// TIA Portal V15.1 export
// export: Created 2024-06-21T08:41:18.3279413Z, ExportSetting WithDefaults, DisplayName Totally Integrated Automation Portal, DisplayVersion V15.1 Update 5, DisplayName TIA Portal Openness, DisplayVersion V15.1 Update 5, DisplayName SINAMICS Startdrive Advanced, DisplayVersion V15.1, DisplayName G130, G150, S120, S150, SINAMICS MV, S210, DisplayVersion V15.1, DisplayName G110M, G120, G120C, G120D, G120P, DisplayVersion V15.1, DisplayName STEP 7 Professional, DisplayVersion V15.1 Update 5, DisplayName STEP 7 Safety, DisplayVersion V15.1, DisplayName WinCC Professional, DisplayVersion V15.1 Update 5, DisplayName SIMATIC Visualization Architect, DisplayVersion V15.1
FUNCTION_BLOCK "LGBRoller1W2S-C"   // FB6678, FBD
TITLE = LRoller2W2S-C / LGBRoller1W2S-C
{ S7_Optimized_Access := 'TRUE' }
AUTHOR : VCC
FAMILY : Transpor
VERSION : 0.1
// =============================================================================
// This module is used in Applications when a roller two way two Speed equipped 
// with contactor is needed.
// The roller can support single body tranport and simultanious transport. The 
// roller is equiped with a standard sensor setting (two at the rear and two at 
// the front for high/low Speed transport). 
// The roller shall use standard handshaking signals to accomplish an infeed 
// transfer with the previous transport system and an outfeed with the next 
// transport system (in both directions).
// The roller will support automatic Mode and manual Mode according specific 
// guidelines. All transport rollers shall use the same principle techniques.
// The outfeed will be master over the infeed Alarm "body not in Position" is also 
// generated. All Alarms coming from sub-functions (TrfIn, TrfOut & Motor2W2S-C) 
// or from local Alarm (see above) are summarized to give also the global Alarm A, 
// B, C & D to upper level.
// =============================================================================
// =============================================================================
// This module is used in Applications when a roller one way two Speed equipped 
// with contactor is needed.
// The roller can support single body tranport and simultanious transport. The 
// roller is equiped with a standard sensor setting (two at the rear and two at 
// the front for high/low Speed transport). 
// The roller shall use standard handshaking signals to accomplish an infeed 
// transfer with the previous transport system and an outfeed with the next 
// transport system (in both directions).
// The roller will support automatic Mode and manual Mode according specific 
// guidelines. All transport rollers shall use the same principle techniques.
// The outfeed will be master over the infeed Alarm "body not in Position" is also 
// generated. All Alarms coming from sub-functions (TrfIn, TrfOut & Motor1W2S-C) 
// or from local Alarm (see above) are summarized to give also the global Alarm A, 
// B, C & D to upper level.
// =============================================================================
// stored: AutoNumber false, IsIECCheckEnabled false, IsRetainMemResEnabled false, MemoryReserve 100, SetENOAutomatically False, UDAEnableTagReadback false
   VAR_INPUT
      I_StopDetSet { ExternalAccessible := 'False'; ExternalVisible := 'False'; ExternalWritable := 'False'} : Bool;   // Stop Detection set
      I_LowSpeedDetSet { ExternalAccessible := 'False'; ExternalVisible := 'False'; ExternalWritable := 'False'} : Bool;   // Lowspeed Detection set
      I_StopDetRes { ExternalAccessible := 'False'; ExternalVisible := 'False'; ExternalWritable := 'False'} : Bool;   // Stop Detection Reset
      I_OccupiedDet { ExternalAccessible := 'False'; ExternalVisible := 'False'; ExternalWritable := 'False'} : Bool;   // Occupied detection
      I_BrakeReleased { ExternalAccessible := 'False'; ExternalVisible := 'False'; ExternalWritable := 'False'} : Bool;   // Feedback from brake contactor
      I_TrfInSetBegin { ExternalAccessible := 'False'; ExternalVisible := 'False'; ExternalWritable := 'False'} : Bool;   // Load Begin: condition to start transfer IN set
      I_TrfInSetIntlkOk { ExternalAccessible := 'False'; ExternalVisible := 'False'; ExternalWritable := 'False'} : Bool;   // Transfer IN Interlock Set OK
      I_TrfOutSetBegin { ExternalAccessible := 'False'; ExternalVisible := 'False'; ExternalWritable := 'False'} : Bool;   // Unload Begin: condition to start transfer OUT set
      I_TrfOutSetIntlkOk { ExternalAccessible := 'False'; ExternalVisible := 'False'; ExternalWritable := 'False'} : Bool;   // Transfer Out Interlock Set Ok
      I_TrfInSetRdyDlv { ExternalAccessible := 'False'; ExternalVisible := 'False'; ExternalWritable := 'False'} : Bool;   // Ready to deliver: Signal from previous object set
      I_TrfInSetTM { ExternalAccessible := 'False'; ExternalVisible := 'False'; ExternalWritable := 'False'} : Bool;   // Transfer busy signal from previous equipement set
      I_TrfOutSetRdyRcv { ExternalAccessible := 'False'; ExternalVisible := 'False'; ExternalWritable := 'False'} : Bool;   // Ready to Receive: Signal from next object set
      I_TrfOutSetArrived { ExternalAccessible := 'False'; ExternalVisible := 'False'; ExternalWritable := 'False'} : Bool;   // Body Arrived: Signal from next object Set
      I_LocalPBSet { ExternalAccessible := 'False'; ExternalVisible := 'False'; ExternalWritable := 'False'} : Bool;   // Push button for manual movememt (on local panel) set
      I_ManInfeedAllowedSet { ExternalAccessible := 'False'; ExternalVisible := 'False'; ExternalWritable := 'False'} : Bool;   // Manual Infeed Allowed Set (without PushButton)
      I_ManLowSpdSel { ExternalAccessible := 'False'; ExternalVisible := 'False'; ExternalWritable := 'False'} : Bool;   // Low speed Selected in manual / Low speed Selected in manual by other roller
      I_ManHighSpdSel { ExternalAccessible := 'False'; ExternalVisible := 'False'; ExternalWritable := 'False'} : Bool;   // Low speed Selected in manual / High speed Selected in manual by other roller
      I_MotorProtection { ExternalAccessible := 'False'; ExternalVisible := 'False'; ExternalWritable := 'False'} : Bool;   // Motorprotection / Motor protection
      I_BrakeProtection { ExternalAccessible := 'False'; ExternalVisible := 'False'; ExternalWritable := 'False'} : Bool;   // Brake protection
      I_SafetySwitch { ExternalAccessible := 'False'; ExternalVisible := 'False'; ExternalWritable := 'False'} : Bool;   // Safety switch
      I_SafetyOk { ExternalAccessible := 'False'; ExternalVisible := 'False'; ExternalWritable := 'False'} : Bool;   // Safety Ok
      I_MotionStopOk { ExternalAccessible := 'False'; ExternalVisible := 'False'; ExternalWritable := 'False'} : Bool;   // Safety Ok / The motion stop is Ok
   END_VAR
   VAR_OUTPUT
      O_ContactorLSpdSet { ExternalAccessible := 'False'; ExternalVisible := 'False'; ExternalWritable := 'False'} : Bool;   // Activate low speed contactor
      O_ContactorHSpdSet { ExternalAccessible := 'False'; ExternalVisible := 'False'; ExternalWritable := 'False'} : Bool;   // Activate High Speed contactor
      O_ReleaseBrakeContactor { ExternalAccessible := 'False'; ExternalVisible := 'False'; ExternalWritable := 'False'} : Bool;   // Release Brake
      O_Active { ExternalAccessible := 'False'; ExternalVisible := 'False'; ExternalWritable := 'False'} : Bool;   // Roller is Active
      O_TrfInSetRdyRcv { ExternalAccessible := 'False'; ExternalVisible := 'False'; ExternalWritable := 'False'} : Bool;   // Ready to Receive: Signal to previous object set
      O_TrfInSetArrived { ExternalAccessible := 'False'; ExternalVisible := 'False'; ExternalWritable := 'False'} : Bool;   // Body Arrived: Signal to previous object Set
      O_TrfOutSetRdyDlv { ExternalAccessible := 'False'; ExternalVisible := 'False'; ExternalWritable := 'False'} : Bool;   // Ready to Deliver: Signal to next object set
      O_TrfOutSetTM { ExternalAccessible := 'False'; ExternalVisible := 'False'; ExternalWritable := 'False'} : Bool;   // Transfer: Signal to next object set
      O_TrfInSetActive { ExternalAccessible := 'False'; ExternalVisible := 'False'; ExternalWritable := 'False'} : Bool;   // Transfer in set active
      O_TrfInSetFinished { ExternalAccessible := 'False'; ExternalVisible := 'False'; ExternalWritable := 'False'} : Bool;   // Transfer in set finished
      O_TrfOutSetActive { ExternalAccessible := 'False'; ExternalVisible := 'False'; ExternalWritable := 'False'} : Bool;   // Transfer out set active
      O_TrfOutSetFinished { ExternalAccessible := 'False'; ExternalVisible := 'False'; ExternalWritable := 'False'} : Bool;   // Transfer out set finished
      O_BodyInPosition { ExternalAccessible := 'False'; ExternalVisible := 'False'; ExternalWritable := 'False'} : Bool;   // Body in Position on roller
      O_ManLowSpdSel { ExternalAccessible := 'False'; ExternalVisible := 'False'; ExternalWritable := 'False'} : Bool;   // Low speed Selected in manual
      O_ManHighSpdSel { ExternalAccessible := 'False'; ExternalVisible := 'False'; ExternalWritable := 'False'} : Bool;   // Low speed Selected in manual / High speed Selected in manual
      O_LedRoller { ExternalAccessible := 'False'; ExternalVisible := 'False'; ExternalWritable := 'False'} : Bool;   // Led of roller
      O_AlarmABCondition { ExternalAccessible := 'False'; ExternalVisible := 'False'; ExternalWritable := 'False'} : Bool;   // Alarm AB Condition
      O_AlarmA { ExternalAccessible := 'False'; ExternalVisible := 'False'; ExternalWritable := 'False'} : Bool;   // Alarm A
      O_AlarmB { ExternalAccessible := 'False'; ExternalVisible := 'False'; ExternalWritable := 'False'} : Bool;   // Alarm B
      O_AlarmC { ExternalAccessible := 'False'; ExternalVisible := 'False'; ExternalWritable := 'False'} : Bool;   // Alarm C
      O_AlarmD { ExternalAccessible := 'False'; ExternalVisible := 'False'; ExternalWritable := 'False'} : Bool;   // Alarm D
      O_Occupied { ExternalAccessible := 'False'; ExternalVisible := 'False'; ExternalWritable := 'False'} : Bool;   // Roller Occupied
      H_AlarmDWord { ExternalAccessible := 'False'; ExternalVisible := 'False'; ExternalWritable := 'False'} : DWord;   // HMI Animation
   END_VAR
   VAR_IN_OUT
      IO_Modes : "Modes";   // Modes
      H_HMI : "H_HMI";   // Animation
      "H_GBRoller1W2S-C" : "H_GBRoller1W2S-C";   // Animation
      C_Config : "RollerConvConfig";   // Config
   END_VAR
   VAR
      AlarmABCondition { ExternalAccessible := 'False'; ExternalVisible := 'False'; ExternalWritable := 'False'} : Bool;   // Alarm AB condition / Alarm AB Condition
      AC_BodyNotInPos { ExternalAccessible := 'False'; ExternalVisible := 'False'; ExternalWritable := 'False'} : Bool;   // Body, Skid Not In Position / Kaross , Skid Ej I Position
      AB_TrfOutSetOverTime { ExternalAccessible := 'False'; ExternalVisible := 'False'; ExternalWritable := 'False'} : Bool;   // Timeout Transport Out Set / Tidsövervakning Uttransport Set
      AD_TrfOutSetInterlock { ExternalAccessible := 'False'; ExternalVisible := 'False'; ExternalWritable := 'False'} : Bool;   // Interlock Not Ok Transport Out Set / Interlock Ej Ok Uttransport Set
      AD_TrfInSetInterlock { ExternalAccessible := 'False'; ExternalVisible := 'False'; ExternalWritable := 'False'} : Bool;   // Interlock Not Ok Transport In Set / Interlock Ej Ok Intransport Set
      AB_LSpeedDetMissing { ExternalAccessible := 'False'; ExternalVisible := 'False'; ExternalWritable := 'False'} : Bool;   // Low Speed Detector Missing / Lågfartsgivare Saknas
      AA_MotorProtector { ExternalAccessible := 'False'; ExternalVisible := 'False'; ExternalWritable := 'False'} : Bool;   // Motorprotection Tripped / Motor Protection Tripped / Motorskydd Utlöst
      AA_BrakeProtector { ExternalAccessible := 'False'; ExternalVisible := 'False'; ExternalWritable := 'False'} : Bool;   // Brake Protection Tripped
      AA_SafetySwitch { ExternalAccessible := 'False'; ExternalVisible := 'False'; ExternalWritable := 'False'} : Bool;   // Safety Switch Not Ok / Säkerhetsbrytare Ej Ok
      AB_BrakeFbk { ExternalAccessible := 'False'; ExternalVisible := 'False'; ExternalWritable := 'False'} : Bool;   // Safety Switch Not Ok / Brake feedback Nok / Säkerhetsbrytare Ej Ok
      AD_MotionStop { ExternalAccessible := 'False'; ExternalVisible := 'False'; ExternalWritable := 'False'} : Bool;   // Motion Stop
      AC_ConfigCalibrationAlm { ExternalAccessible := 'False'; ExternalVisible := 'False'; ExternalWritable := 'False'} : Bool;   // The Config values for Alarm Transfer time must be ALL zero or ALL different from zero
      AD_CalibrationSetWarn { ExternalAccessible := 'False'; ExternalVisible := 'False'; ExternalWritable := 'False'} : Bool;   // No High speed selected so Calibration is not possible for SET direction
      SafetyOk { ExternalAccessible := 'False'; ExternalVisible := 'False'; ExternalWritable := 'False'} : Bool;   // Safety Ok
      LowSpeedSetDetOk { ExternalAccessible := 'False'; ExternalVisible := 'False'; ExternalWritable := 'False'} : Bool;   // Low speed detector set ok
      AllDet { ExternalAccessible := 'False'; ExternalVisible := 'False'; ExternalWritable := 'False'} : Bool;   // AND of ALL detections
      AnyDet { ExternalAccessible := 'False'; ExternalVisible := 'False'; ExternalWritable := 'False'} : Bool;   // OR of ALL Detections
      MotorLoopActive { ExternalAccessible := 'False'; ExternalVisible := 'False'; ExternalWritable := 'False'} : Bool;   // Motor Loop Active
      TrfInSetIntlkOk { ExternalAccessible := 'False'; ExternalVisible := 'False'; ExternalWritable := 'False'} : Bool;   // Transfer IN Interlock Set OK
      TrfOutSetIntlkOk { ExternalAccessible := 'False'; ExternalVisible := 'False'; ExternalWritable := 'False'} : Bool;   // Transfer Out Interlock Set Ok
      TrfInfeedHoldSet { ExternalAccessible := 'False'; ExternalVisible := 'False'; ExternalWritable := 'False'} : Bool;   // Transfer infeed hold set direction
      TrfOutSetCmd { ExternalAccessible := 'False'; ExternalVisible := 'False'; ExternalWritable := 'False'} : Bool;   // Command after Interlock to Motor set
      TrfOutfeedHoldSet { ExternalAccessible := 'False'; ExternalVisible := 'False'; ExternalWritable := 'False'} : Bool;   // Transfer outfeed hold set direction
      TrfInSetCmd { ExternalAccessible := 'False'; ExternalVisible := 'False'; ExternalWritable := 'False'} : Bool;   // Command after Interlock to Motor set
      MotorCmdLSpdSet { ExternalAccessible := 'False'; ExternalVisible := 'False'; ExternalWritable := 'False'} : Bool;   // Command to Motorloop low Speed Set
      MotorCmdHSpdSet { ExternalAccessible := 'False'; ExternalVisible := 'False'; ExternalWritable := 'False'} : Bool;   // Command to Motorloop High Speed Set
      LowSpeedDetSetMem { ExternalAccessible := 'False'; ExternalVisible := 'False'; ExternalWritable := 'False'} : Bool;   // memorisation stop High Speed Set direction
      TrfInSetActive { ExternalAccessible := 'False'; ExternalVisible := 'False'; ExternalWritable := 'False'} : Bool;   // Load: Active (set)
      TrfOutSetActive { ExternalAccessible := 'False'; ExternalVisible := 'False'; ExternalWritable := 'False'} : Bool;   // Unload: active (set)
      TrfOutSetFinished { ExternalAccessible := 'False'; ExternalVisible := 'False'; ExternalWritable := 'False'} : Bool;   // Unload: finished (set)
      AlarmA { ExternalAccessible := 'False'; ExternalVisible := 'False'; ExternalWritable := 'False'} : Bool;   // Alarm A
      AlarmB { ExternalAccessible := 'False'; ExternalVisible := 'False'; ExternalWritable := 'False'} : Bool;   // Alarm B
      AlarmC { ExternalAccessible := 'False'; ExternalVisible := 'False'; ExternalWritable := 'False'} : Bool;   // Alarm C
      AlarmD { ExternalAccessible := 'False'; ExternalVisible := 'False'; ExternalWritable := 'False'} : Bool;   // Alarm D
      ManLowSpdSel { ExternalAccessible := 'False'; ExternalVisible := 'False'; ExternalWritable := 'False'} : Bool;   // Low speed Selected in manual
      BodyInPosition { ExternalAccessible := 'False'; ExternalVisible := 'False'; ExternalWritable := 'False'} : Bool;   // Body in Position
      TrfOutSetRdyDlv { ExternalAccessible := 'False'; ExternalVisible := 'False'; ExternalWritable := 'False'} : Bool;   // Ready to Deliver: Signal to next object set
      TrfOutSetTM { ExternalAccessible := 'False'; ExternalVisible := 'False'; ExternalWritable := 'False'} : Bool;   // Transfer : Signal transfer memory to next object set
      TrfInSetTrfOutSetTM { ExternalAccessible := 'False'; ExternalVisible := 'False'; ExternalWritable := 'False'} : Bool;   // Transfer memory set
      TrfInSetRdyRcv { ExternalAccessible := 'False'; ExternalVisible := 'False'; ExternalWritable := 'False'} : Bool;   // Ready to Receive: Signal to previous object set
      TrfInSetArrived { ExternalAccessible := 'False'; ExternalVisible := 'False'; ExternalWritable := 'False'} : Bool;   // Body Arrived: Signal to previous object Set
      TrfInSetFinished { ExternalAccessible := 'False'; ExternalVisible := 'False'; ExternalWritable := 'False'} : Bool;   // Body Arrived: Signal to TrfOut module set (Reset TrfOutCmd)
      StopTrfOutSetCmd { ExternalAccessible := 'False'; ExternalVisible := 'False'; ExternalWritable := 'False'} : Bool;   // Body Arrived: Signal to previous object Set
      MotorLoopAlmCond { ExternalAccessible := 'False'; ExternalVisible := 'False'; ExternalWritable := 'False'} : Bool;   // Motor loop Alarm condition
      TrfOutSetAlmCond { ExternalAccessible := 'False'; ExternalVisible := 'False'; ExternalWritable := 'False'} : Bool;   // TrfOut set Alarm condition
      ContactorLSpdSet { ExternalAccessible := 'False'; ExternalVisible := 'False'; ExternalWritable := 'False'} : Bool;   // Contactor low speed
      ContactorHSpdSet { ExternalAccessible := 'False'; ExternalVisible := 'False'; ExternalWritable := 'False'} : Bool;   // Contactor High Speed
      ReleaseBrakeContactor { ExternalAccessible := 'False'; ExternalVisible := 'False'; ExternalWritable := 'False'} : Bool;   // Activate Reset contactor / Release Brake contactor
      LowSpeedDetMisingCond { ExternalAccessible := 'False'; ExternalVisible := 'False'; ExternalWritable := 'False'} : Bool;   // Low speed detector misiing condition
      _LTrfInSet { ExternalAccessible := 'False'; ExternalVisible := 'False'; ExternalWritable := 'False'} : "LGBTrfIn";   // FB
      _LTrfOutSet { ExternalAccessible := 'False'; ExternalVisible := 'False'; ExternalWritable := 'False'} : "LGBTrfOut";   // FB
      _Motor { ExternalAccessible := 'False'; ExternalVisible := 'False'; ExternalWritable := 'False'} : "LGBMotor1W2S-C";   // FB
   END_VAR
   VAR_TEMP
      H_HMITrfInSet : "H_HMI";   // Temp
      H_HMITrfOutSet : "H_HMI";   // Temp
      H_HMIMotor : "H_HMI";   // Temp
   END_VAR
   VAR_TEMP   // added for the SCL form of the ladder/FBD networks
      _w1 : Bool;
   END_VAR
BEGIN

REGION Network 1: **** 1 - Inputs **** AND of all detections
   // AND of all detections
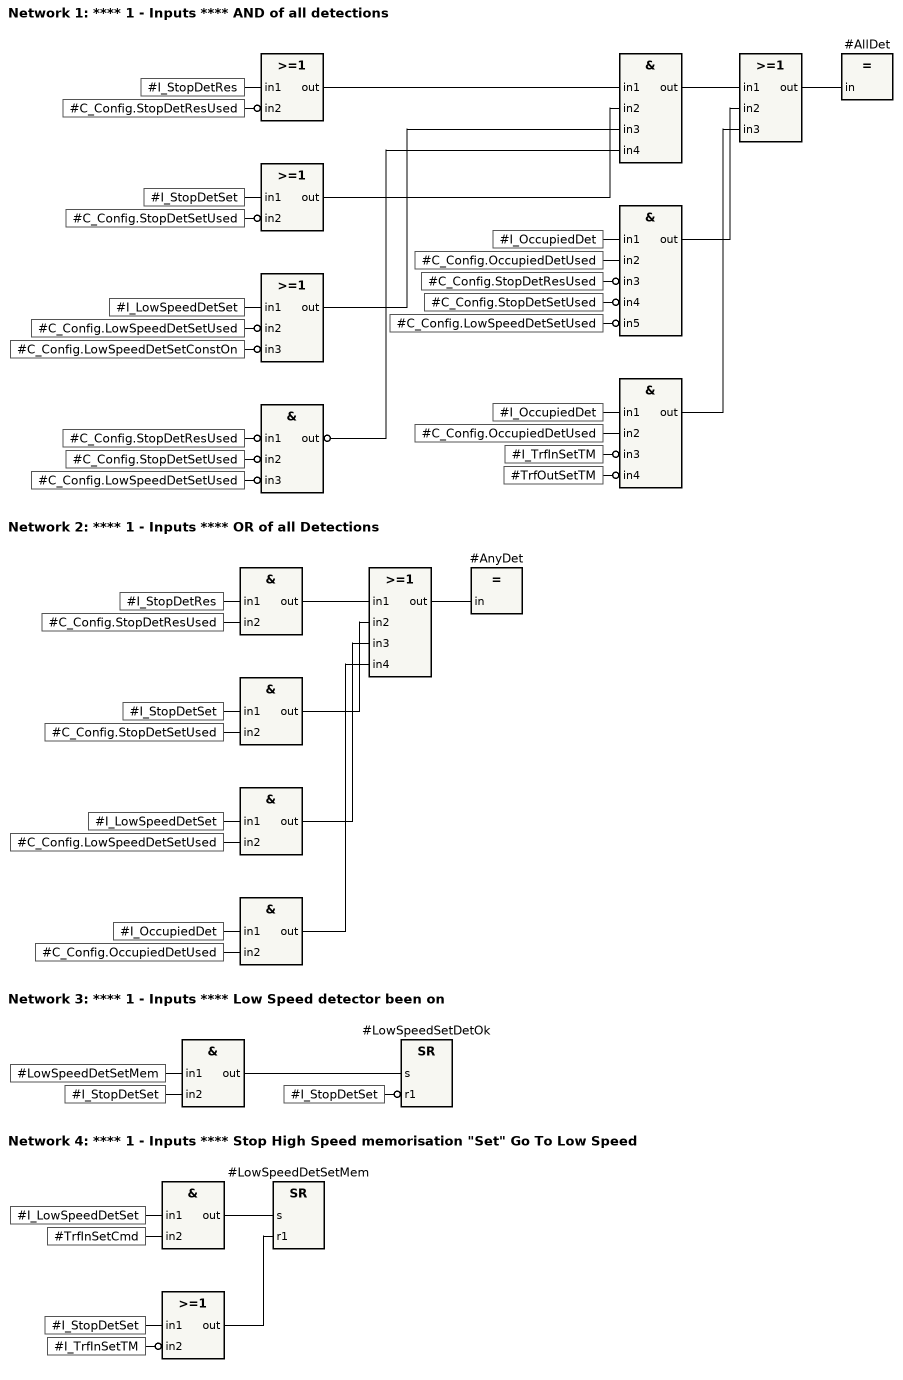
   #AllDet := ((#I_StopDetRes OR NOT #C_Config.StopDetResUsed) AND (#I_StopDetSet OR NOT #C_Config.StopDetSetUsed) AND (#I_LowSpeedDetSet OR NOT #C_Config.LowSpeedDetSetUsed OR NOT #C_Config.LowSpeedDetSetConstOn) AND NOT (NOT #C_Config.StopDetResUsed AND NOT #C_Config.StopDetSetUsed AND NOT #C_Config.LowSpeedDetSetUsed)) OR (#I_OccupiedDet AND #C_Config.OccupiedDetUsed AND NOT #C_Config.StopDetResUsed AND NOT #C_Config.StopDetSetUsed AND NOT #C_Config.LowSpeedDetSetUsed) OR (#I_OccupiedDet AND #C_Config.OccupiedDetUsed AND NOT #I_TrfInSetTM AND NOT #TrfOutSetTM);
END_REGION

REGION Network 2: **** 1 - Inputs **** OR of all Detections
   // OR of all Detections
   #AnyDet := (#I_StopDetRes AND #C_Config.StopDetResUsed) OR (#I_StopDetSet AND #C_Config.StopDetSetUsed) OR (#I_LowSpeedDetSet AND #C_Config.LowSpeedDetSetUsed) OR (#I_OccupiedDet AND #C_Config.OccupiedDetUsed);
END_REGION

REGION Network 3: **** 1 - Inputs **** Low Speed detector been on
   // Low Speed detector been on
   IF #LowSpeedDetSetMem AND #I_StopDetSet THEN
       #LowSpeedSetDetOk := TRUE;   // SR flip-flop
   END_IF;
   IF NOT #I_StopDetSet THEN #LowSpeedSetDetOk := FALSE; END_IF;
END_REGION

REGION Network 4: **** 1 - Inputs **** Stop High Speed memorisation "Set" Go To Low Speed
   // Stop High Speed memorisation (set) (go to low Speed)
   IF #I_LowSpeedDetSet AND #TrfInSetCmd THEN
       #LowSpeedDetSetMem := TRUE;   // SR flip-flop
   END_IF;
   IF #I_StopDetSet OR NOT #I_TrfInSetTM THEN #LowSpeedDetSetMem := FALSE; END_IF;
END_REGION

REGION Network 5: **** 1 - Inputs **** Transfer IN Interlock Set OK
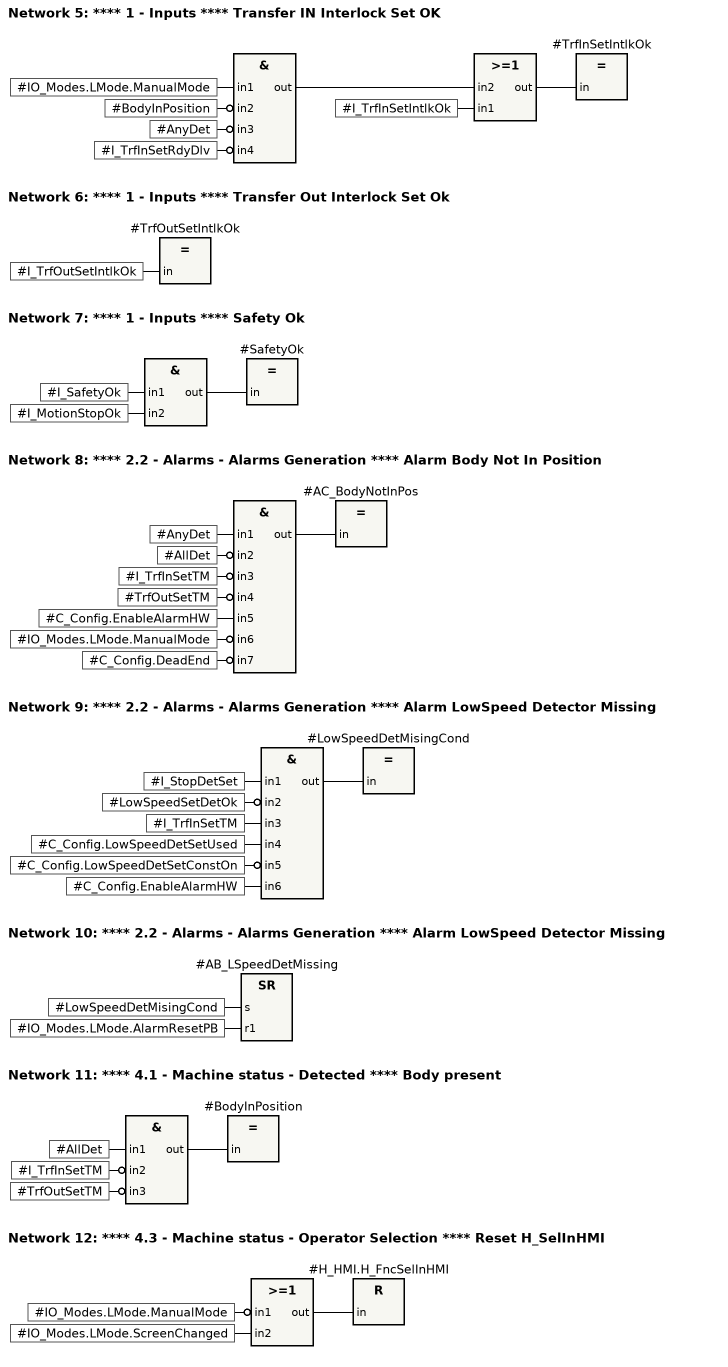
   #TrfInSetIntlkOk := (#IO_Modes.LMode.ManualMode AND NOT #BodyInPosition AND NOT #AnyDet AND NOT #I_TrfInSetRdyDlv) OR #I_TrfInSetIntlkOk;
END_REGION

REGION Network 6: **** 1 - Inputs **** Transfer Out Interlock Set Ok
   #TrfOutSetIntlkOk := #I_TrfOutSetIntlkOk;
END_REGION

REGION Network 7: **** 1 - Inputs **** Safety Ok
   #SafetyOk := #I_SafetyOk AND #I_MotionStopOk;
END_REGION

REGION Network 8: **** 2.2 - Alarms - Alarms Generation **** Alarm Body Not In Position
   // Alarm Body Not In Position
   #AC_BodyNotInPos := #AnyDet AND NOT #AllDet AND NOT #I_TrfInSetTM AND NOT #TrfOutSetTM AND #C_Config.EnableAlarmHW AND NOT #IO_Modes.LMode.ManualMode AND NOT #C_Config.DeadEnd;
END_REGION

REGION Network 9: **** 2.2 - Alarms - Alarms Generation **** Alarm LowSpeed Detector Missing
   // Alarm LowSpeed Detector Missing
   #LowSpeedDetMisingCond := #I_StopDetSet AND NOT #LowSpeedSetDetOk AND #I_TrfInSetTM AND #C_Config.LowSpeedDetSetUsed AND NOT #C_Config.LowSpeedDetSetConstOn AND #C_Config.EnableAlarmHW;
END_REGION

REGION Network 10: **** 2.2 - Alarms - Alarms Generation **** Alarm LowSpeed Detector Missing
   // Alarm LowSpeed Detector Missing
   IF #LowSpeedDetMisingCond THEN
       #AB_LSpeedDetMissing := TRUE;   // SR flip-flop
   END_IF;
   IF #IO_Modes.LMode.AlarmResetPB THEN #AB_LSpeedDetMissing := FALSE; END_IF;
END_REGION

REGION Network 11: **** 4.1 - Machine status - Detected **** Body present
   // Body present
   #BodyInPosition := #AllDet AND NOT #I_TrfInSetTM AND NOT #TrfOutSetTM;
END_REGION

REGION Network 12: **** 4.3 - Machine status - Operator Selection **** Reset H_SelInHMI
   // Reset H_SelInHMI
   IF NOT #IO_Modes.LMode.ManualMode OR #IO_Modes.LMode.ScreenChanged THEN
       #H_HMI.H_FncSelInHMI := FALSE;
   END_IF;
END_REGION

REGION Network 13: **** 4.6 - Machine status - Indications **** Active
   // Active
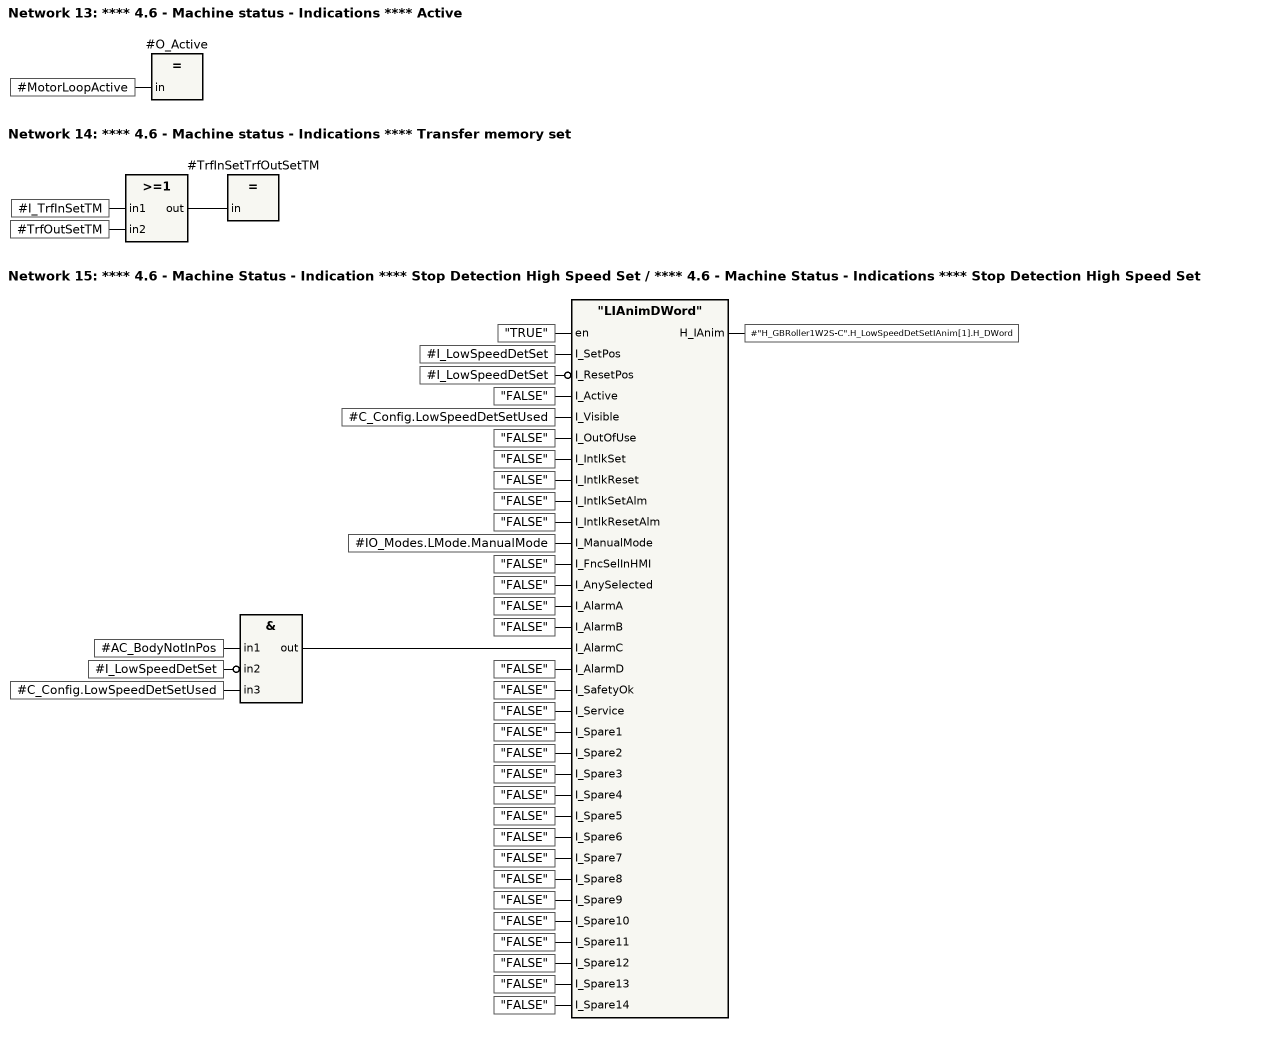
   #O_Active := #MotorLoopActive;
END_REGION

REGION Network 14: **** 4.6 - Machine status - Indications **** Transfer memory set
   // Transfer memory set
   #TrfInSetTrfOutSetTM := #I_TrfInSetTM OR #TrfOutSetTM;
END_REGION

REGION Network 15: **** 4.6 - Machine Status - Indication **** Stop Detection High Speed Set / **** 4.6 - Machine Status - Indications **** Stop Detection High Speed Set
   // Stop Detection High Speed Set
   IF "TRUE" THEN
       "LIAnimDWord"(I_SetPos := #I_LowSpeedDetSet,
                     I_ResetPos := NOT #I_LowSpeedDetSet,
                     I_Active := "FALSE",
                     I_Visible := #C_Config.LowSpeedDetSetUsed,
                     I_OutOfUse := "FALSE",
                     I_IntlkSet := "FALSE",
                     I_IntlkReset := "FALSE",
                     I_IntlkSetAlm := "FALSE",
                     I_IntlkResetAlm := "FALSE",
                     I_ManualMode := #IO_Modes.LMode.ManualMode,
                     I_FncSelInHMI := "FALSE",
                     I_AnySelected := "FALSE",
                     I_AlarmA := "FALSE",
                     I_AlarmB := "FALSE",
                     I_AlarmC := #AC_BodyNotInPos AND NOT #I_LowSpeedDetSet AND #C_Config.LowSpeedDetSetUsed,
                     I_AlarmD := "FALSE",
                     I_SafetyOk := "FALSE",
                     I_Service := "FALSE",
                     I_Spare1 := "FALSE",
                     I_Spare2 := "FALSE",
                     I_Spare3 := "FALSE",
                     I_Spare4 := "FALSE",
                     I_Spare5 := "FALSE",
                     I_Spare6 := "FALSE",
                     I_Spare7 := "FALSE",
                     I_Spare8 := "FALSE",
                     I_Spare9 := "FALSE",
                     I_Spare10 := "FALSE",
                     I_Spare11 := "FALSE",
                     I_Spare12 := "FALSE",
                     I_Spare13 := "FALSE",
                     I_Spare14 := "FALSE",
                     H_IAnim => #"H_GBRoller1W2S-C".H_LowSpeedDetSetIAnim[1].H_DWord);
   END_IF;
END_REGION

REGION Network 16: **** 4.6 - Machine Status - Indication **** Stop Detection set / **** 4.6 - Machine Status - Indications **** Stop Detection set
   // Stop Detection set
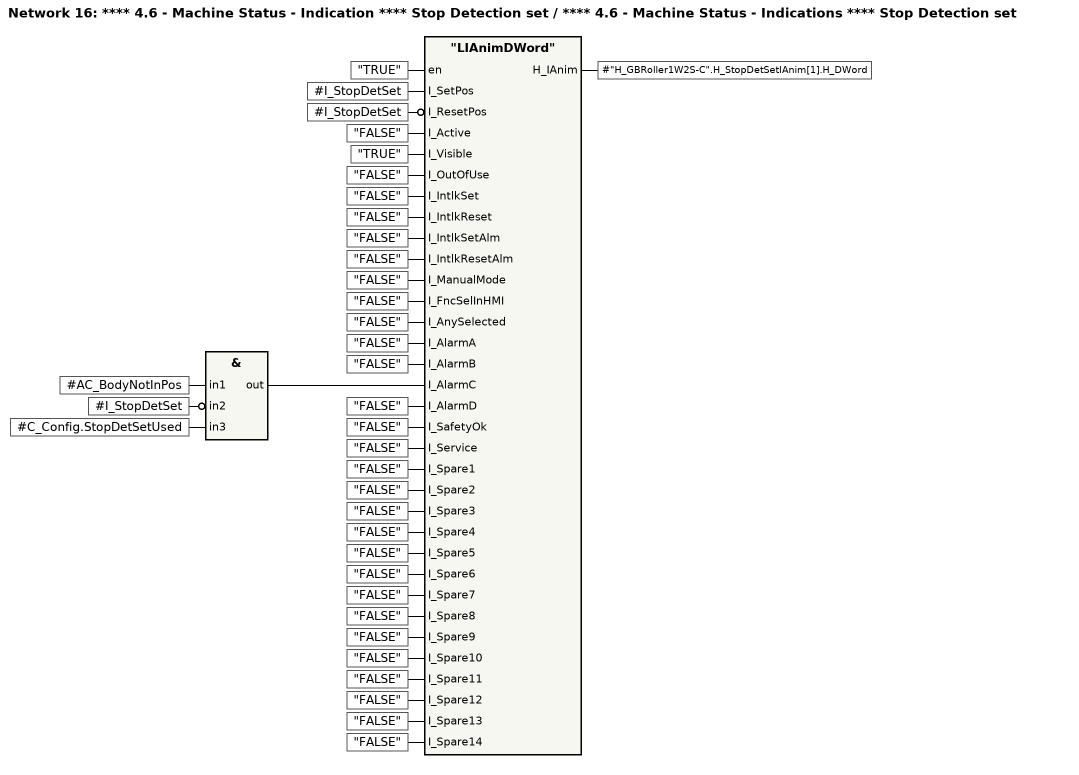
   IF "TRUE" THEN
       "LIAnimDWord"(I_SetPos := #I_StopDetSet,
                     I_ResetPos := NOT #I_StopDetSet,
                     I_Active := "FALSE",
                     I_Visible := "TRUE",
                     I_OutOfUse := "FALSE",
                     I_IntlkSet := "FALSE",
                     I_IntlkReset := "FALSE",
                     I_IntlkSetAlm := "FALSE",
                     I_IntlkResetAlm := "FALSE",
                     I_ManualMode := "FALSE",
                     I_FncSelInHMI := "FALSE",
                     I_AnySelected := "FALSE",
                     I_AlarmA := "FALSE",
                     I_AlarmB := "FALSE",
                     I_AlarmC := #AC_BodyNotInPos AND NOT #I_StopDetSet AND #C_Config.StopDetSetUsed,
                     I_AlarmD := "FALSE",
                     I_SafetyOk := "FALSE",
                     I_Service := "FALSE",
                     I_Spare1 := "FALSE",
                     I_Spare2 := "FALSE",
                     I_Spare3 := "FALSE",
                     I_Spare4 := "FALSE",
                     I_Spare5 := "FALSE",
                     I_Spare6 := "FALSE",
                     I_Spare7 := "FALSE",
                     I_Spare8 := "FALSE",
                     I_Spare9 := "FALSE",
                     I_Spare10 := "FALSE",
                     I_Spare11 := "FALSE",
                     I_Spare12 := "FALSE",
                     I_Spare13 := "FALSE",
                     I_Spare14 := "FALSE",
                     H_IAnim => #"H_GBRoller1W2S-C".H_StopDetSetIAnim[1].H_DWord);
   END_IF;
END_REGION

REGION Network 17: **** 4.6 - Machine Status - Indication **** Stop Detection Reset / **** 4.6 - Machine Status - Indications **** Stop Detection Reset
   // Stop Detection Reset
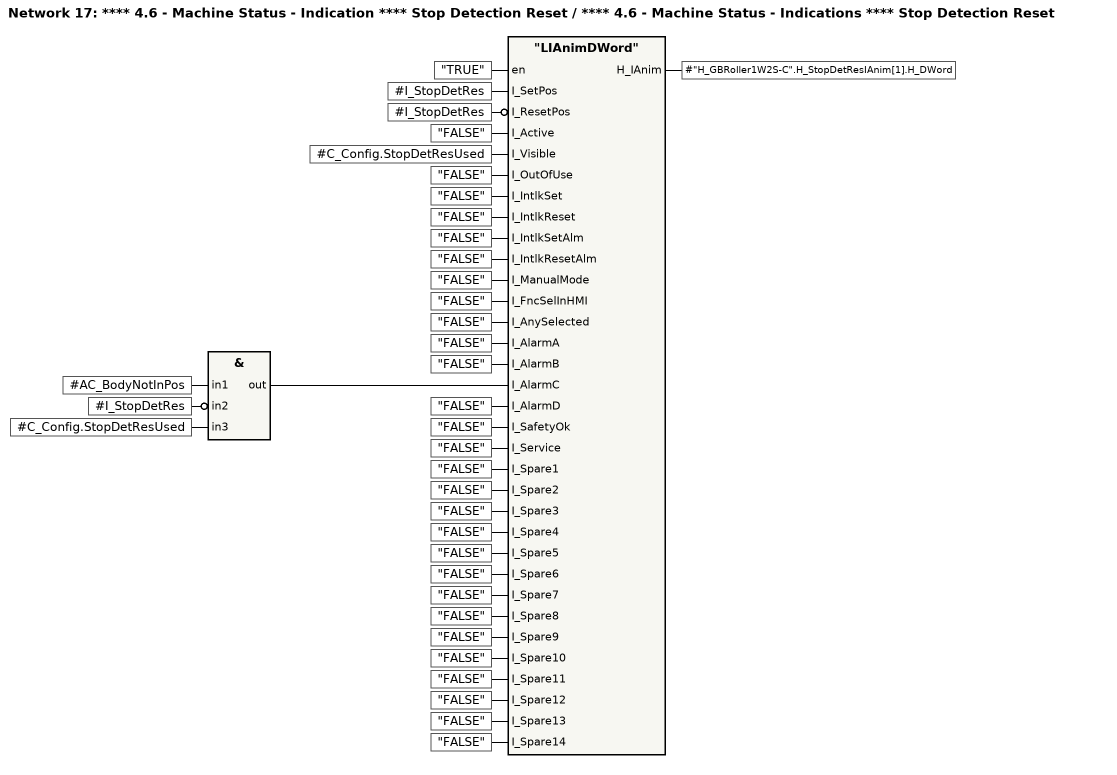
   IF "TRUE" THEN
       "LIAnimDWord"(I_SetPos := #I_StopDetRes,
                     I_ResetPos := NOT #I_StopDetRes,
                     I_Active := "FALSE",
                     I_Visible := #C_Config.StopDetResUsed,
                     I_OutOfUse := "FALSE",
                     I_IntlkSet := "FALSE",
                     I_IntlkReset := "FALSE",
                     I_IntlkSetAlm := "FALSE",
                     I_IntlkResetAlm := "FALSE",
                     I_ManualMode := "FALSE",
                     I_FncSelInHMI := "FALSE",
                     I_AnySelected := "FALSE",
                     I_AlarmA := "FALSE",
                     I_AlarmB := "FALSE",
                     I_AlarmC := #AC_BodyNotInPos AND NOT #I_StopDetRes AND #C_Config.StopDetResUsed,
                     I_AlarmD := "FALSE",
                     I_SafetyOk := "FALSE",
                     I_Service := "FALSE",
                     I_Spare1 := "FALSE",
                     I_Spare2 := "FALSE",
                     I_Spare3 := "FALSE",
                     I_Spare4 := "FALSE",
                     I_Spare5 := "FALSE",
                     I_Spare6 := "FALSE",
                     I_Spare7 := "FALSE",
                     I_Spare8 := "FALSE",
                     I_Spare9 := "FALSE",
                     I_Spare10 := "FALSE",
                     I_Spare11 := "FALSE",
                     I_Spare12 := "FALSE",
                     I_Spare13 := "FALSE",
                     I_Spare14 := "FALSE",
                     H_IAnim => #"H_GBRoller1W2S-C".H_StopDetResIAnim[1].H_DWord);
   END_IF;
END_REGION

REGION Network 18: **** 4.6 - Machine Status - Indication **** Stop Detection Reset / **** 4.6 - Machine Status - Indication **** Occupied Detection
   // Stop detection Reset / Occupied Detection
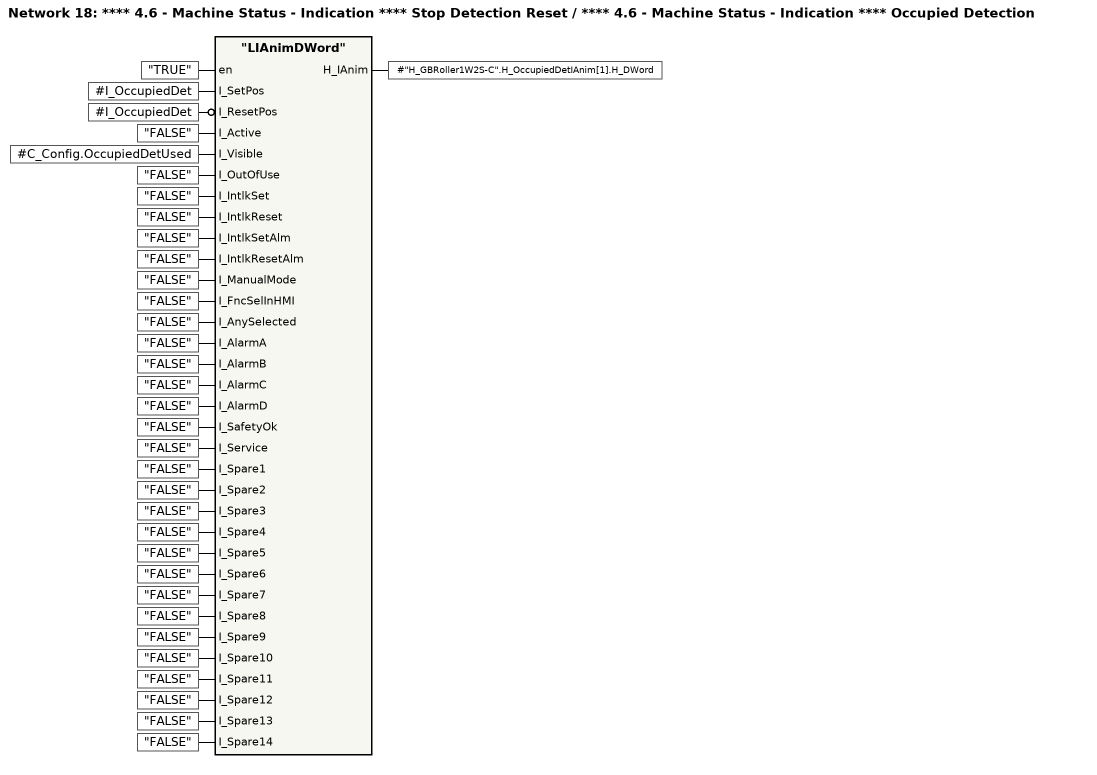
   IF "TRUE" THEN
       "LIAnimDWord"(I_SetPos := #I_OccupiedDet,
                     I_ResetPos := NOT #I_OccupiedDet,
                     I_Active := "FALSE",
                     I_Visible := #C_Config.OccupiedDetUsed,
                     I_OutOfUse := "FALSE",
                     I_IntlkSet := "FALSE",
                     I_IntlkReset := "FALSE",
                     I_IntlkSetAlm := "FALSE",
                     I_IntlkResetAlm := "FALSE",
                     I_ManualMode := "FALSE",
                     I_FncSelInHMI := "FALSE",
                     I_AnySelected := "FALSE",
                     I_AlarmA := "FALSE",
                     I_AlarmB := "FALSE",
                     I_AlarmC := "FALSE",
                     I_AlarmD := "FALSE",
                     I_SafetyOk := "FALSE",
                     I_Service := "FALSE",
                     I_Spare1 := "FALSE",
                     I_Spare2 := "FALSE",
                     I_Spare3 := "FALSE",
                     I_Spare4 := "FALSE",
                     I_Spare5 := "FALSE",
                     I_Spare6 := "FALSE",
                     I_Spare7 := "FALSE",
                     I_Spare8 := "FALSE",
                     I_Spare9 := "FALSE",
                     I_Spare10 := "FALSE",
                     I_Spare11 := "FALSE",
                     I_Spare12 := "FALSE",
                     I_Spare13 := "FALSE",
                     I_Spare14 := "FALSE",
                     H_IAnim => #"H_GBRoller1W2S-C".H_OccupiedDetIAnim[1].H_DWord);
   END_IF;
END_REGION

REGION Network 19: **** 4.6 - Machine Status - Indication **** Icon Animation / **** 4.6 - Machine Status - Indications **** Icon Animation
   // Icon Animation
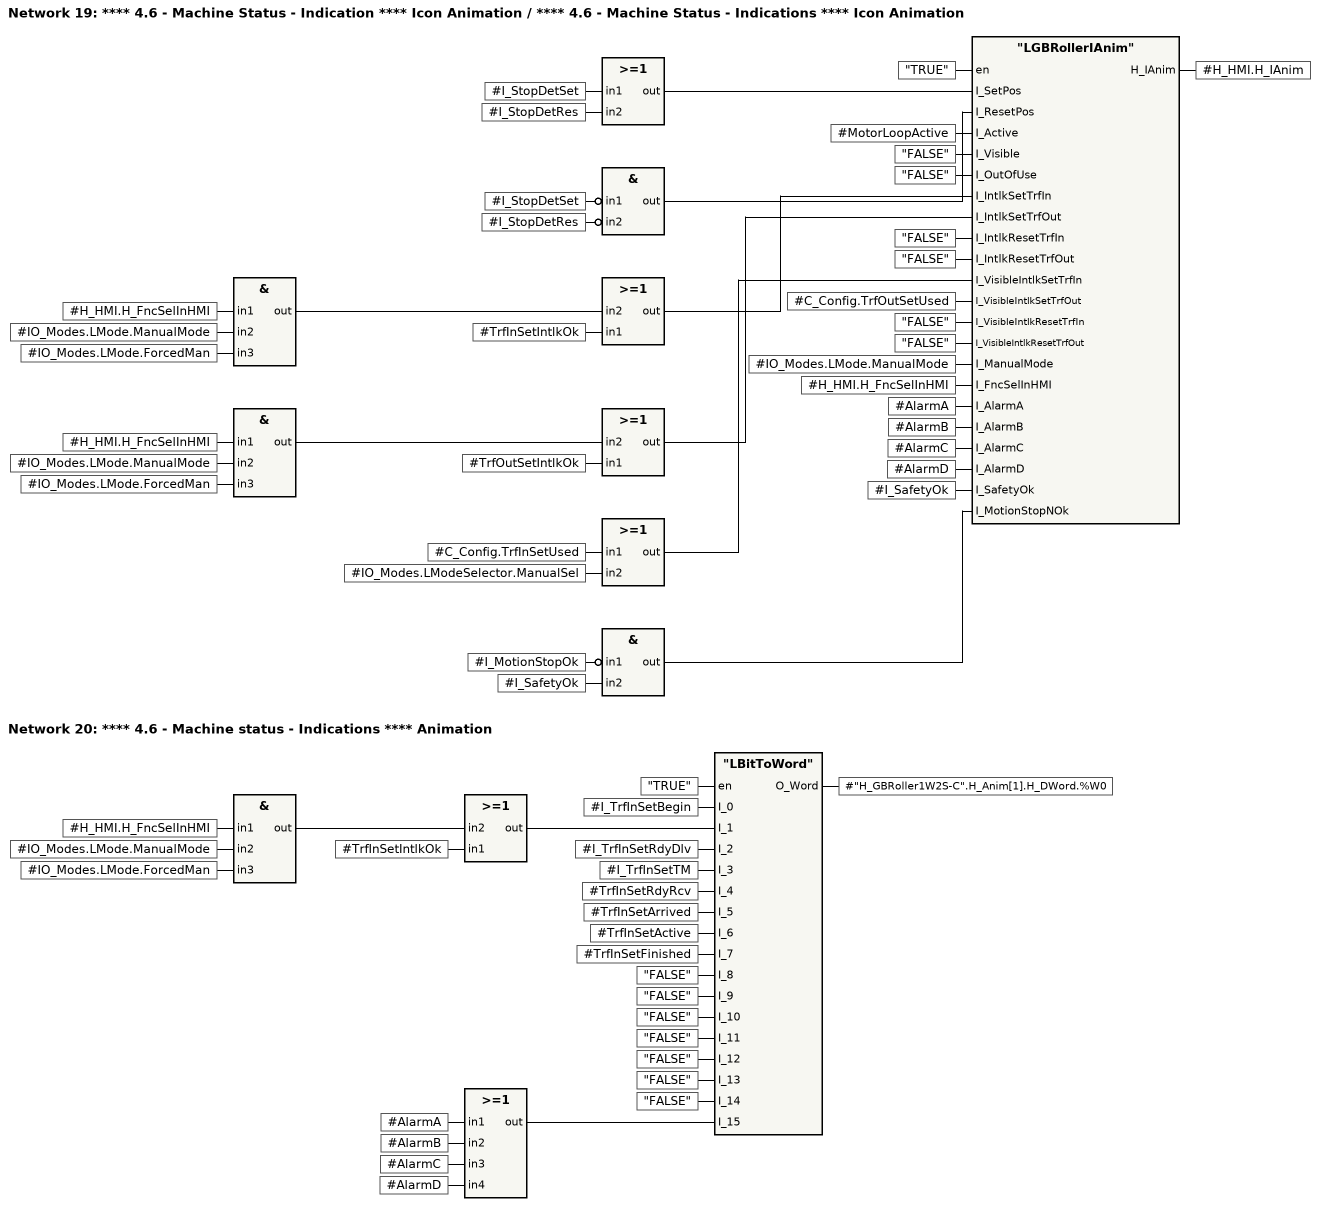
   IF "TRUE" THEN
       "LGBRollerIAnim"(I_SetPos := #I_StopDetSet OR #I_StopDetRes,
                        I_ResetPos := NOT #I_StopDetSet AND NOT #I_StopDetRes,
                        I_Active := #MotorLoopActive,
                        I_Visible := "FALSE",
                        I_OutOfUse := "FALSE",
                        I_IntlkSetTrfIn := (#H_HMI.H_FncSelInHMI AND #IO_Modes.LMode.ManualMode AND #IO_Modes.LMode.ForcedMan) OR #TrfInSetIntlkOk,
                        I_IntlkSetTrfOut := (#H_HMI.H_FncSelInHMI AND #IO_Modes.LMode.ManualMode AND #IO_Modes.LMode.ForcedMan) OR #TrfOutSetIntlkOk,
                        I_IntlkResetTrfIn := "FALSE",
                        I_IntlkResetTrfOut := "FALSE",
                        I_VisibleIntlkSetTrfIn := #C_Config.TrfInSetUsed OR #IO_Modes.LModeSelector.ManualSel,
                        I_VisibleIntlkSetTrfOut := #C_Config.TrfOutSetUsed,
                        I_VisibleIntlkResetTrfIn := "FALSE",
                        I_VisibleIntlkResetTrfOut := "FALSE",
                        I_ManualMode := #IO_Modes.LMode.ManualMode,
                        I_FncSelInHMI := #H_HMI.H_FncSelInHMI,
                        I_AlarmA := #AlarmA,
                        I_AlarmB := #AlarmB,
                        I_AlarmC := #AlarmC,
                        I_AlarmD := #AlarmD,
                        I_SafetyOk := #I_SafetyOk,
                        I_MotionStopNOk := NOT #I_MotionStopOk AND #I_SafetyOk,
                        H_IAnim => #H_HMI.H_IAnim);
   END_IF;
END_REGION

REGION Network 20: **** 4.6 - Machine status - Indications **** Animation
   // Animation
   IF "TRUE" THEN
       "LBitToWord"(I_0 := #I_TrfInSetBegin,
                    I_1 := (#H_HMI.H_FncSelInHMI AND #IO_Modes.LMode.ManualMode AND #IO_Modes.LMode.ForcedMan) OR #TrfInSetIntlkOk,
                    I_2 := #I_TrfInSetRdyDlv,
                    I_3 := #I_TrfInSetTM,
                    I_4 := #TrfInSetRdyRcv,
                    I_5 := #TrfInSetArrived,
                    I_6 := #TrfInSetActive,
                    I_7 := #TrfInSetFinished,
                    I_8 := "FALSE",
                    I_9 := "FALSE",
                    I_10 := "FALSE",
                    I_11 := "FALSE",
                    I_12 := "FALSE",
                    I_13 := "FALSE",
                    I_14 := "FALSE",
                    I_15 := #AlarmA OR #AlarmB OR #AlarmC OR #AlarmD,
                    O_Word => #"H_GBRoller1W2S-C".H_Anim[1].H_DWord.%W0);
   END_IF;
END_REGION

REGION Network 21: **** 4.6 - Machine status - Indications **** Animation
   // Animation
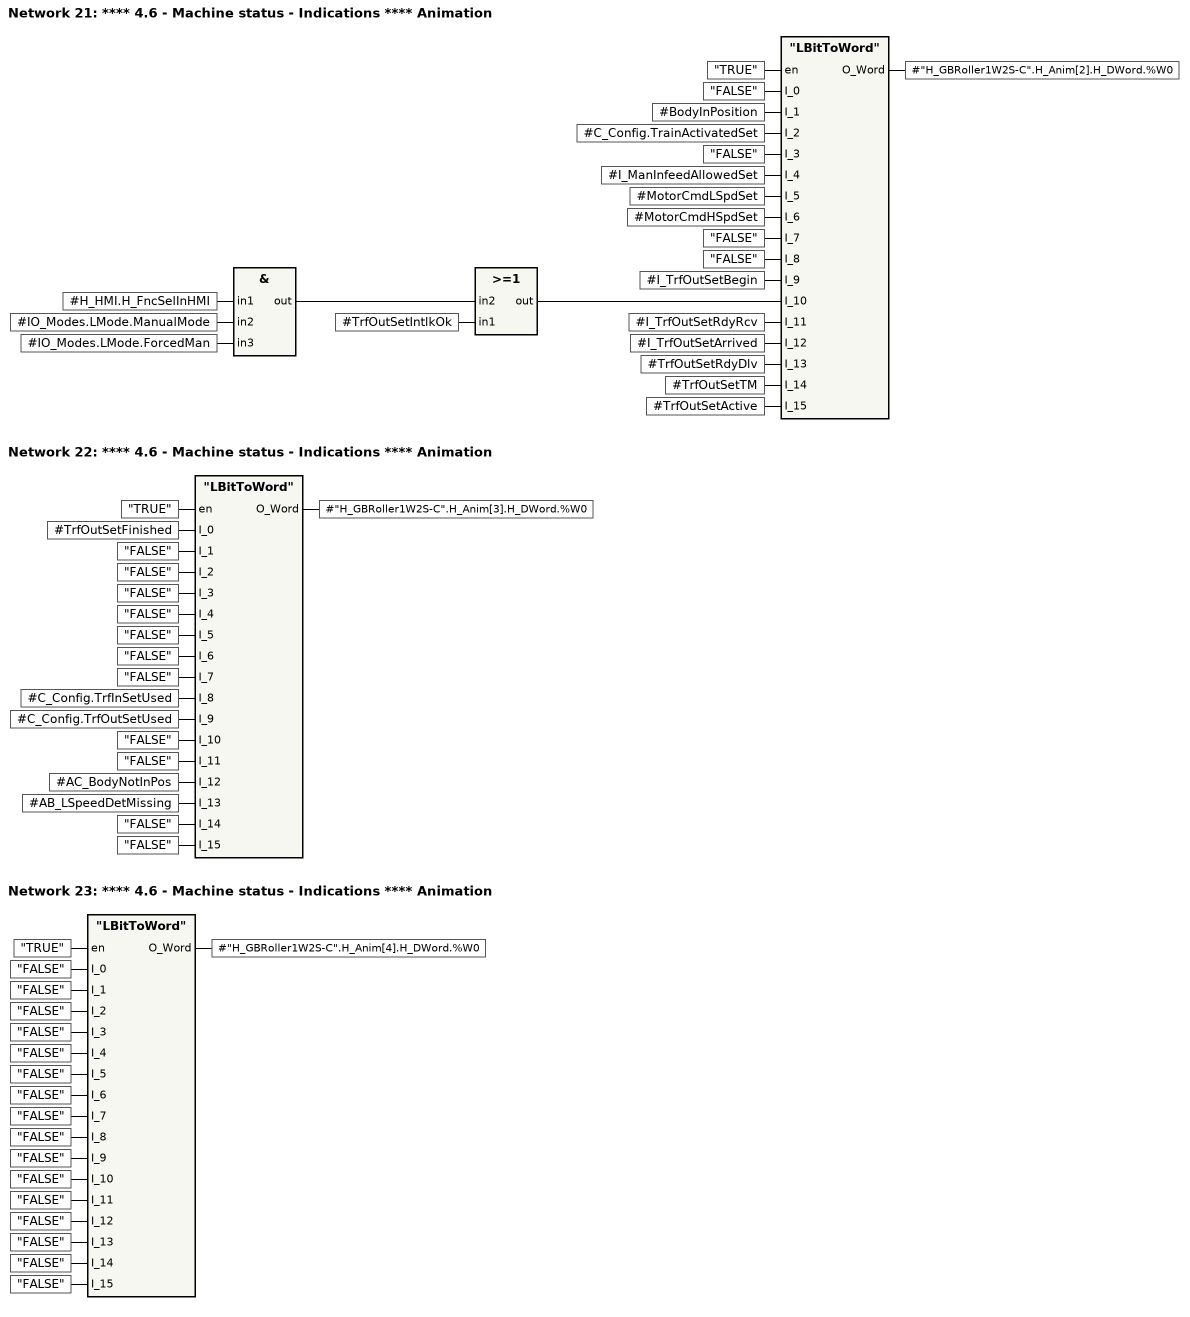
   IF "TRUE" THEN
       "LBitToWord"(I_0 := "FALSE",
                    I_1 := #BodyInPosition,
                    I_2 := #C_Config.TrainActivatedSet,
                    I_3 := "FALSE",
                    I_4 := #I_ManInfeedAllowedSet,
                    I_5 := #MotorCmdLSpdSet,
                    I_6 := #MotorCmdHSpdSet,
                    I_7 := "FALSE",
                    I_8 := "FALSE",
                    I_9 := #I_TrfOutSetBegin,
                    I_10 := (#H_HMI.H_FncSelInHMI AND #IO_Modes.LMode.ManualMode AND #IO_Modes.LMode.ForcedMan) OR #TrfOutSetIntlkOk,
                    I_11 := #I_TrfOutSetRdyRcv,
                    I_12 := #I_TrfOutSetArrived,
                    I_13 := #TrfOutSetRdyDlv,
                    I_14 := #TrfOutSetTM,
                    I_15 := #TrfOutSetActive,
                    O_Word => #"H_GBRoller1W2S-C".H_Anim[2].H_DWord.%W0);
   END_IF;
END_REGION

REGION Network 22: **** 4.6 - Machine status - Indications **** Animation
   // Animation
   IF "TRUE" THEN
       "LBitToWord"(I_0 := #TrfOutSetFinished,
                    I_1 := "FALSE",
                    I_2 := "FALSE",
                    I_3 := "FALSE",
                    I_4 := "FALSE",
                    I_5 := "FALSE",
                    I_6 := "FALSE",
                    I_7 := "FALSE",
                    I_8 := #C_Config.TrfInSetUsed,
                    I_9 := #C_Config.TrfOutSetUsed,
                    I_10 := "FALSE",
                    I_11 := "FALSE",
                    I_12 := #AC_BodyNotInPos,
                    I_13 := #AB_LSpeedDetMissing,
                    I_14 := "FALSE",
                    I_15 := "FALSE",
                    O_Word => #"H_GBRoller1W2S-C".H_Anim[3].H_DWord.%W0);
   END_IF;
END_REGION

REGION Network 23: **** 4.6 - Machine status - Indications **** Animation
   // Animation
   IF "TRUE" THEN
       "LBitToWord"(I_0 := "FALSE",
                    I_1 := "FALSE",
                    I_2 := "FALSE",
                    I_3 := "FALSE",
                    I_4 := "FALSE",
                    I_5 := "FALSE",
                    I_6 := "FALSE",
                    I_7 := "FALSE",
                    I_8 := "FALSE",
                    I_9 := "FALSE",
                    I_10 := "FALSE",
                    I_11 := "FALSE",
                    I_12 := "FALSE",
                    I_13 := "FALSE",
                    I_14 := "FALSE",
                    I_15 := "FALSE",
                    O_Word => #"H_GBRoller1W2S-C".H_Anim[4].H_DWord.%W0);
   END_IF;
END_REGION

REGION Network 24: **** 7.1 - Submodule - Non-Machine **** Transfer IN Set
   // Transfer IN Set
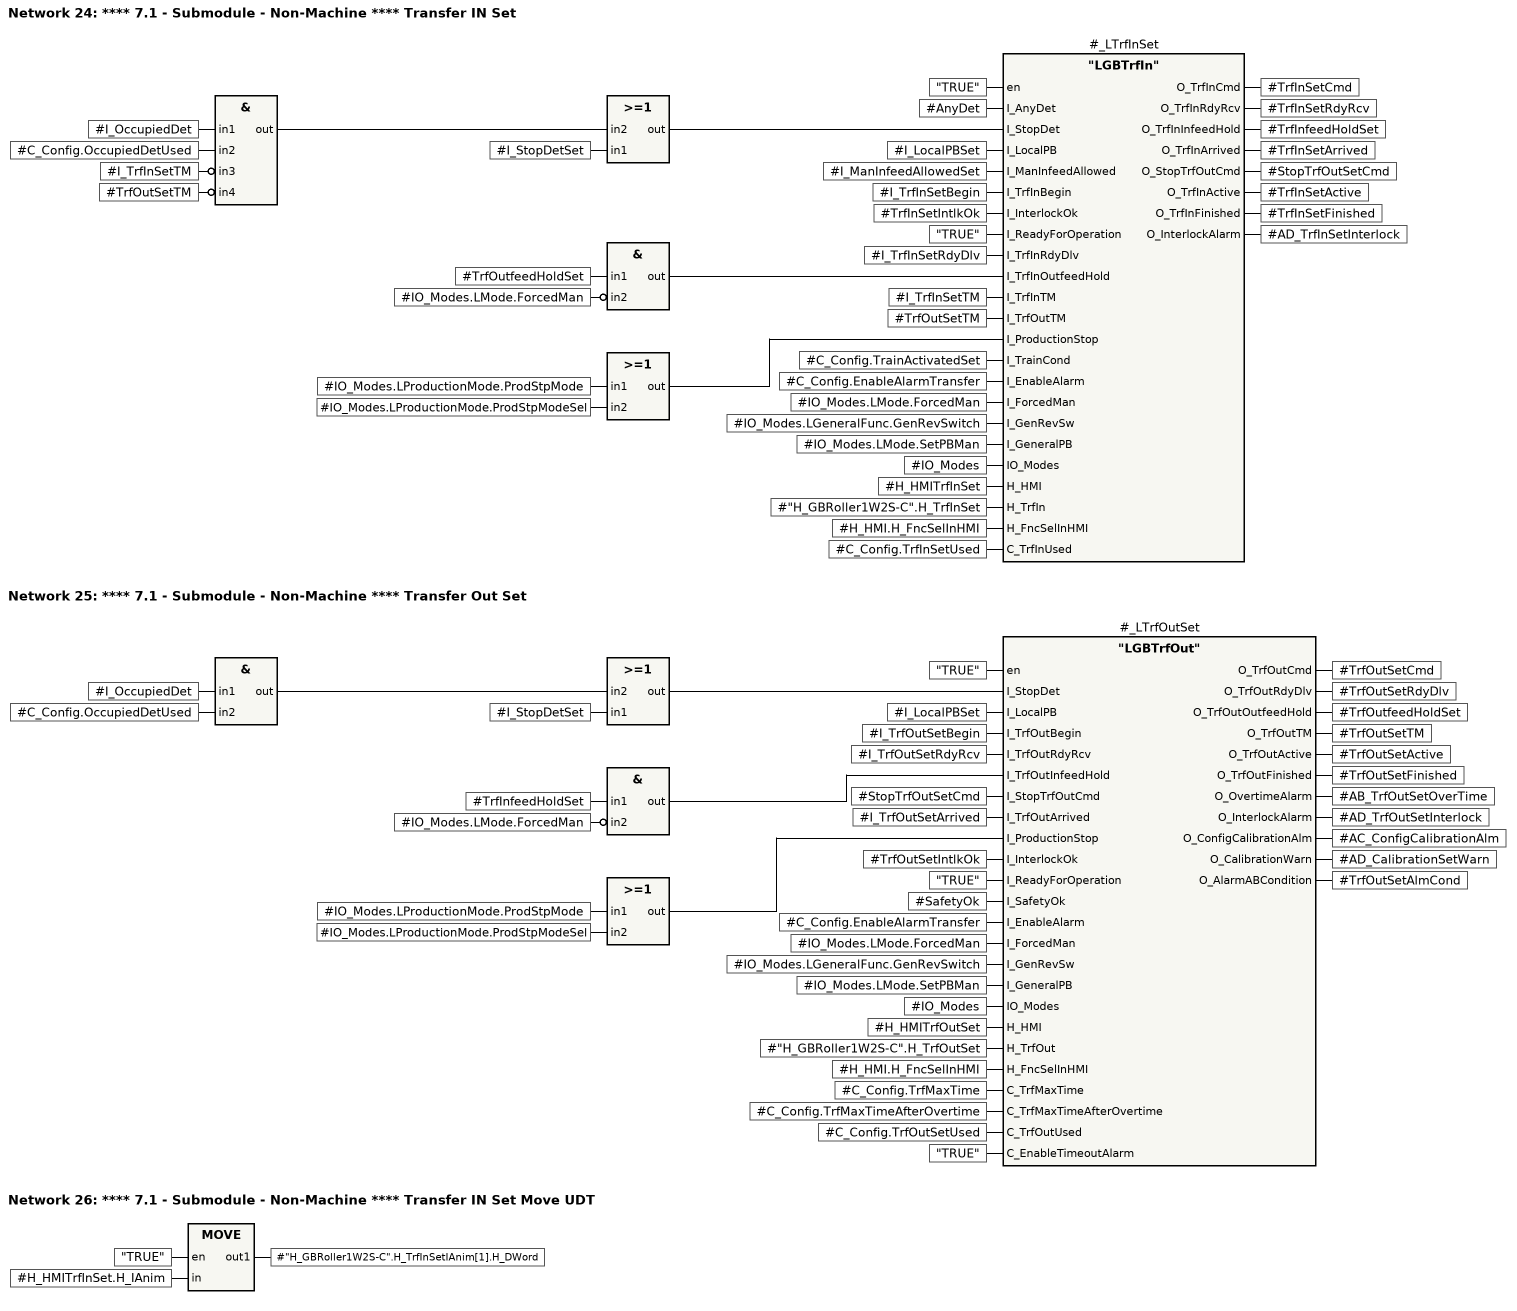
   IF "TRUE" THEN
       #_LTrfInSet(I_AnyDet := #AnyDet,   // "LGBTrfIn"
                   I_StopDet := (#I_OccupiedDet AND #C_Config.OccupiedDetUsed AND NOT #I_TrfInSetTM AND NOT #TrfOutSetTM) OR #I_StopDetSet,
                   I_LocalPB := #I_LocalPBSet,
                   I_ManInfeedAllowed := #I_ManInfeedAllowedSet,
                   I_TrfInBegin := #I_TrfInSetBegin,
                   I_InterlockOk := #TrfInSetIntlkOk,
                   I_ReadyForOperation := "TRUE",
                   I_TrfInRdyDlv := #I_TrfInSetRdyDlv,
                   I_TrfInOutfeedHold := #TrfOutfeedHoldSet AND NOT #IO_Modes.LMode.ForcedMan,
                   I_TrfInTM := #I_TrfInSetTM,
                   I_TrfOutTM := #TrfOutSetTM,
                   I_ProductionStop := #IO_Modes.LProductionMode.ProdStpMode OR #IO_Modes.LProductionMode.ProdStpModeSel,
                   I_TrainCond := #C_Config.TrainActivatedSet,
                   I_EnableAlarm := #C_Config.EnableAlarmTransfer,
                   I_ForcedMan := #IO_Modes.LMode.ForcedMan,
                   I_GenRevSw := #IO_Modes.LGeneralFunc.GenRevSwitch,
                   I_GeneralPB := #IO_Modes.LMode.SetPBMan,
                   IO_Modes := #IO_Modes,
                   H_HMI := #H_HMITrfInSet,
                   H_TrfIn := #"H_GBRoller1W2S-C".H_TrfInSet,
                   H_FncSelInHMI := #H_HMI.H_FncSelInHMI,
                   C_TrfInUsed := #C_Config.TrfInSetUsed,
                   O_TrfInCmd => #TrfInSetCmd,
                   O_TrfInRdyRcv => #TrfInSetRdyRcv,
                   O_TrfInInfeedHold => #TrfInfeedHoldSet,
                   O_TrfInArrived => #TrfInSetArrived,
                   O_StopTrfOutCmd => #StopTrfOutSetCmd,
                   O_TrfInActive => #TrfInSetActive,
                   O_TrfInFinished => #TrfInSetFinished,
                   O_InterlockAlarm => #AD_TrfInSetInterlock);
   END_IF;
END_REGION

REGION Network 25: **** 7.1 - Submodule - Non-Machine **** Transfer Out Set
   // Transfer Out Set
   IF "TRUE" THEN
       #_LTrfOutSet(I_StopDet := (#I_OccupiedDet AND #C_Config.OccupiedDetUsed) OR #I_StopDetSet,   // "LGBTrfOut"
                    I_LocalPB := #I_LocalPBSet,
                    I_TrfOutBegin := #I_TrfOutSetBegin,
                    I_TrfOutRdyRcv := #I_TrfOutSetRdyRcv,
                    I_TrfOutInfeedHold := #TrfInfeedHoldSet AND NOT #IO_Modes.LMode.ForcedMan,
                    I_StopTrfOutCmd := #StopTrfOutSetCmd,
                    I_TrfOutArrived := #I_TrfOutSetArrived,
                    I_ProductionStop := #IO_Modes.LProductionMode.ProdStpMode OR #IO_Modes.LProductionMode.ProdStpModeSel,
                    I_InterlockOk := #TrfOutSetIntlkOk,
                    I_ReadyForOperation := "TRUE",
                    I_SafetyOk := #SafetyOk,
                    I_EnableAlarm := #C_Config.EnableAlarmTransfer,
                    I_ForcedMan := #IO_Modes.LMode.ForcedMan,
                    I_GenRevSw := #IO_Modes.LGeneralFunc.GenRevSwitch,
                    I_GeneralPB := #IO_Modes.LMode.SetPBMan,
                    IO_Modes := #IO_Modes,
                    H_HMI := #H_HMITrfOutSet,
                    H_TrfOut := #"H_GBRoller1W2S-C".H_TrfOutSet,
                    H_FncSelInHMI := #H_HMI.H_FncSelInHMI,
                    C_TrfMaxTime := #C_Config.TrfMaxTime,
                    C_TrfMaxTimeAfterOvertime := #C_Config.TrfMaxTimeAfterOvertime,
                    C_TrfOutUsed := #C_Config.TrfOutSetUsed,
                    C_EnableTimeoutAlarm := "TRUE",
                    O_TrfOutCmd => #TrfOutSetCmd,
                    O_TrfOutRdyDlv => #TrfOutSetRdyDlv,
                    O_TrfOutOutfeedHold => #TrfOutfeedHoldSet,
                    O_TrfOutTM => #TrfOutSetTM,
                    O_TrfOutActive => #TrfOutSetActive,
                    O_TrfOutFinished => #TrfOutSetFinished,
                    O_OvertimeAlarm => #AB_TrfOutSetOverTime,
                    O_InterlockAlarm => #AD_TrfOutSetInterlock,
                    O_ConfigCalibrationAlm => #AC_ConfigCalibrationAlm,
                    O_CalibrationWarn => #AD_CalibrationSetWarn,
                    O_AlarmABCondition => #TrfOutSetAlmCond);
   END_IF;
END_REGION

REGION Network 26: **** 7.1 - Submodule - Non-Machine **** Transfer IN Set Move UDT
   // Transfer IN Set Move UDT
   IF "TRUE" THEN #"H_GBRoller1W2S-C".H_TrfInSetIAnim[1].H_DWord := #H_HMITrfInSet.H_IAnim; END_IF;
END_REGION

REGION Network 27: **** 7.1 - Submodule - Non-Machine **** Transfer Out Set Move UDT
   // Transfer Out Set Move UDT
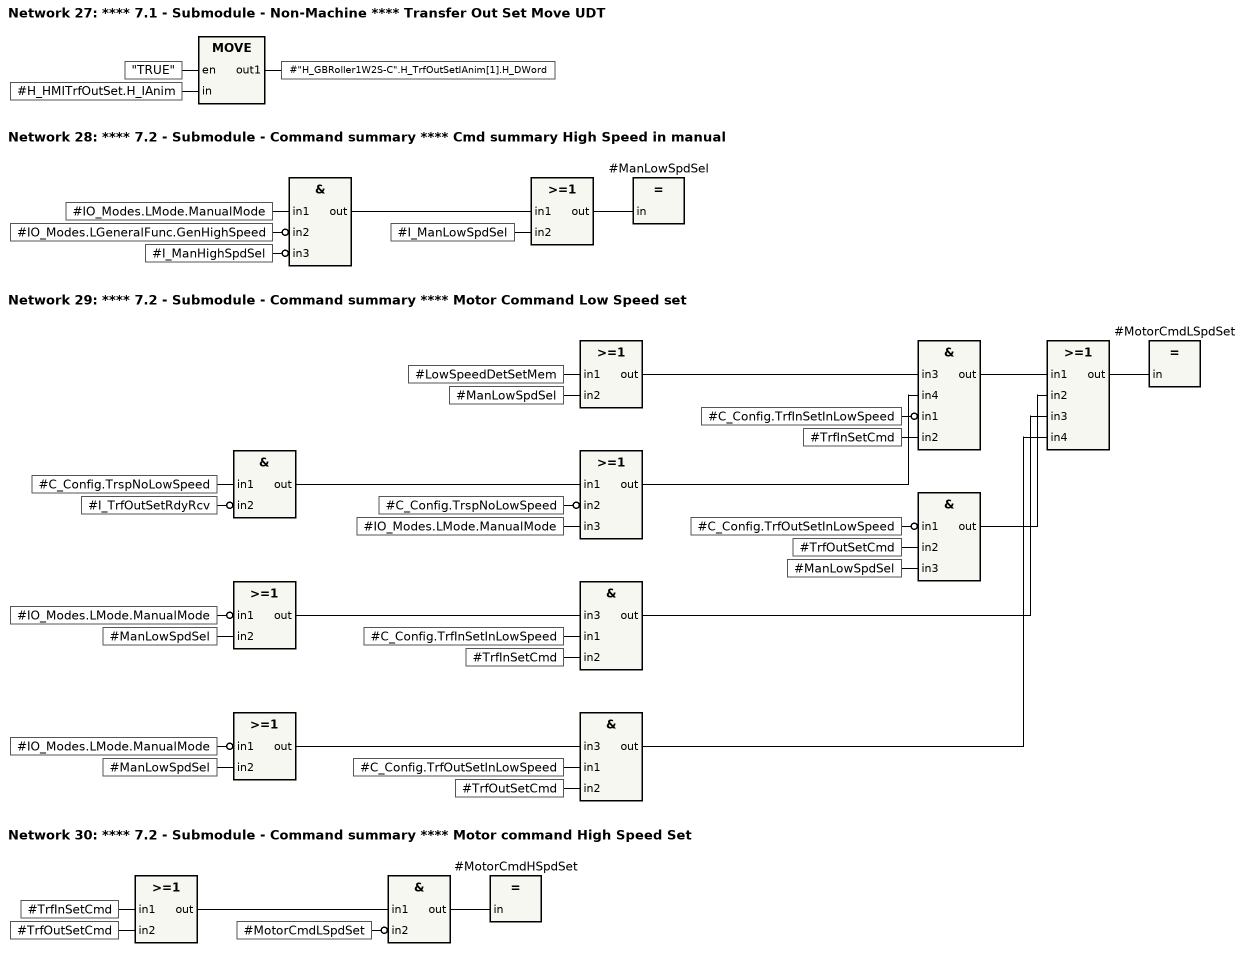
   IF "TRUE" THEN #"H_GBRoller1W2S-C".H_TrfOutSetIAnim[1].H_DWord := #H_HMITrfOutSet.H_IAnim; END_IF;
END_REGION

REGION Network 28: **** 7.2 - Submodule - Command summary **** Cmd summary High Speed in manual
   // Cmd summary High Speed in manual
   #ManLowSpdSel := (#IO_Modes.LMode.ManualMode AND NOT #IO_Modes.LGeneralFunc.GenHighSpeed AND NOT #I_ManHighSpdSel) OR #I_ManLowSpdSel;
END_REGION

REGION Network 29: **** 7.2 - Submodule - Command summary **** Motor Command Low Speed set
   // Motor Command Low Speed Set
   #MotorCmdLSpdSet := ((#LowSpeedDetSetMem OR #ManLowSpdSel) AND ((#C_Config.TrspNoLowSpeed AND NOT #I_TrfOutSetRdyRcv) OR NOT #C_Config.TrspNoLowSpeed OR #IO_Modes.LMode.ManualMode) AND NOT #C_Config.TrfInSetInLowSpeed AND #TrfInSetCmd) OR (NOT #C_Config.TrfOutSetInLowSpeed AND #TrfOutSetCmd AND #ManLowSpdSel) OR ((NOT #IO_Modes.LMode.ManualMode OR #ManLowSpdSel) AND #C_Config.TrfInSetInLowSpeed AND #TrfInSetCmd) OR ((NOT #IO_Modes.LMode.ManualMode OR #ManLowSpdSel) AND #C_Config.TrfOutSetInLowSpeed AND #TrfOutSetCmd);
END_REGION

REGION Network 30: **** 7.2 - Submodule - Command summary **** Motor command High Speed Set
   // Motor command High Speed Set
   #MotorCmdHSpdSet := (#TrfInSetCmd OR #TrfOutSetCmd) AND NOT #MotorCmdLSpdSet;
END_REGION

REGION Network 31: **** 7.3 - Submodule - Machine **** Motor loop
   // Motor loop
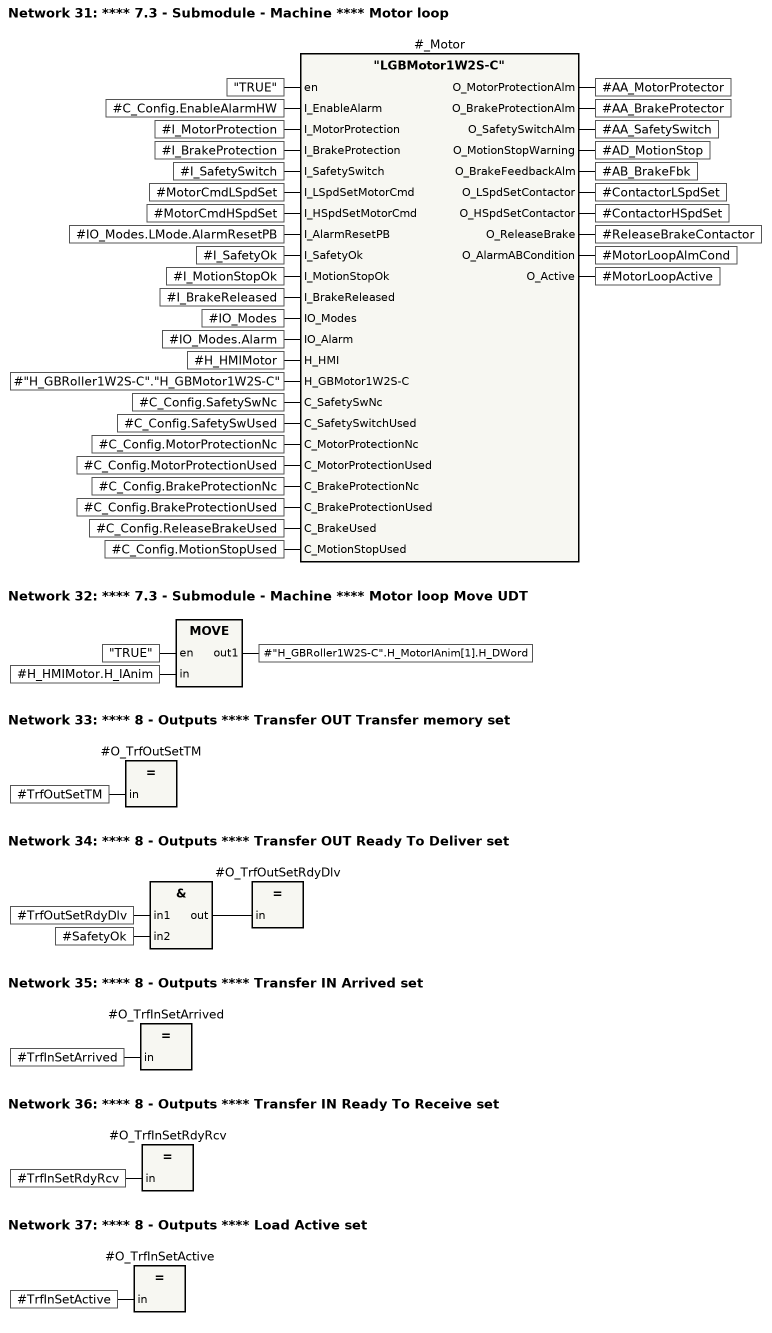
   IF "TRUE" THEN
       #_Motor(I_EnableAlarm := #C_Config.EnableAlarmHW,   // "LGBMotor1W2S-C"
               I_MotorProtection := #I_MotorProtection,
               I_BrakeProtection := #I_BrakeProtection,
               I_SafetySwitch := #I_SafetySwitch,
               I_LSpdSetMotorCmd := #MotorCmdLSpdSet,
               I_HSpdSetMotorCmd := #MotorCmdHSpdSet,
               I_AlarmResetPB := #IO_Modes.LMode.AlarmResetPB,
               I_SafetyOk := #I_SafetyOk,
               I_MotionStopOk := #I_MotionStopOk,
               I_BrakeReleased := #I_BrakeReleased,
               IO_Modes := #IO_Modes,
               IO_Alarm := #IO_Modes.Alarm,
               H_HMI := #H_HMIMotor,
               "H_GBMotor1W2S-C" := #"H_GBRoller1W2S-C"."H_GBMotor1W2S-C",
               C_SafetySwNc := #C_Config.SafetySwNc,
               C_SafetySwitchUsed := #C_Config.SafetySwUsed,
               C_MotorProtectionNc := #C_Config.MotorProtectionNc,
               C_MotorProtectionUsed := #C_Config.MotorProtectionUsed,
               C_BrakeProtectionNc := #C_Config.BrakeProtectionNc,
               C_BrakeProtectionUsed := #C_Config.BrakeProtectionUsed,
               C_BrakeUsed := #C_Config.ReleaseBrakeUsed,
               C_MotionStopUsed := #C_Config.MotionStopUsed,
               O_MotorProtectionAlm => #AA_MotorProtector,
               O_BrakeProtectionAlm => #AA_BrakeProtector,
               O_SafetySwitchAlm => #AA_SafetySwitch,
               O_MotionStopWarning => #AD_MotionStop,
               O_BrakeFeedbackAlm => #AB_BrakeFbk,
               O_LSpdSetContactor => #ContactorLSpdSet,
               O_HSpdSetContactor => #ContactorHSpdSet,
               O_ReleaseBrake => #ReleaseBrakeContactor,
               O_AlarmABCondition => #MotorLoopAlmCond,
               O_Active => #MotorLoopActive);
   END_IF;
END_REGION

REGION Network 32: **** 7.3 - Submodule - Machine **** Motor loop Move UDT
   IF "TRUE" THEN #"H_GBRoller1W2S-C".H_MotorIAnim[1].H_DWord := #H_HMIMotor.H_IAnim; END_IF;
END_REGION

REGION Network 33: **** 8 - Outputs **** Transfer OUT Transfer memory set
   // Transfer OUT Transfer memory set
   #O_TrfOutSetTM := #TrfOutSetTM;
END_REGION

REGION Network 34: **** 8 - Outputs **** Transfer OUT Ready To Deliver set
   // Transfer OUT Ready To Deliver set
   #O_TrfOutSetRdyDlv := #TrfOutSetRdyDlv AND #SafetyOk;
END_REGION

REGION Network 35: **** 8 - Outputs **** Transfer IN Arrived set
   // Transfer IN Arrived set
   #O_TrfInSetArrived := #TrfInSetArrived;
END_REGION

REGION Network 36: **** 8 - Outputs **** Transfer IN Ready To Receive set
   // Transfer IN Ready To Receive set
   #O_TrfInSetRdyRcv := #TrfInSetRdyRcv;
END_REGION

REGION Network 37: **** 8 - Outputs **** Load Active set
   // Load Active set
   #O_TrfInSetActive := #TrfInSetActive;
END_REGION

REGION Network 38: **** 8 - Outputs **** Load finished set
   // Load finished set
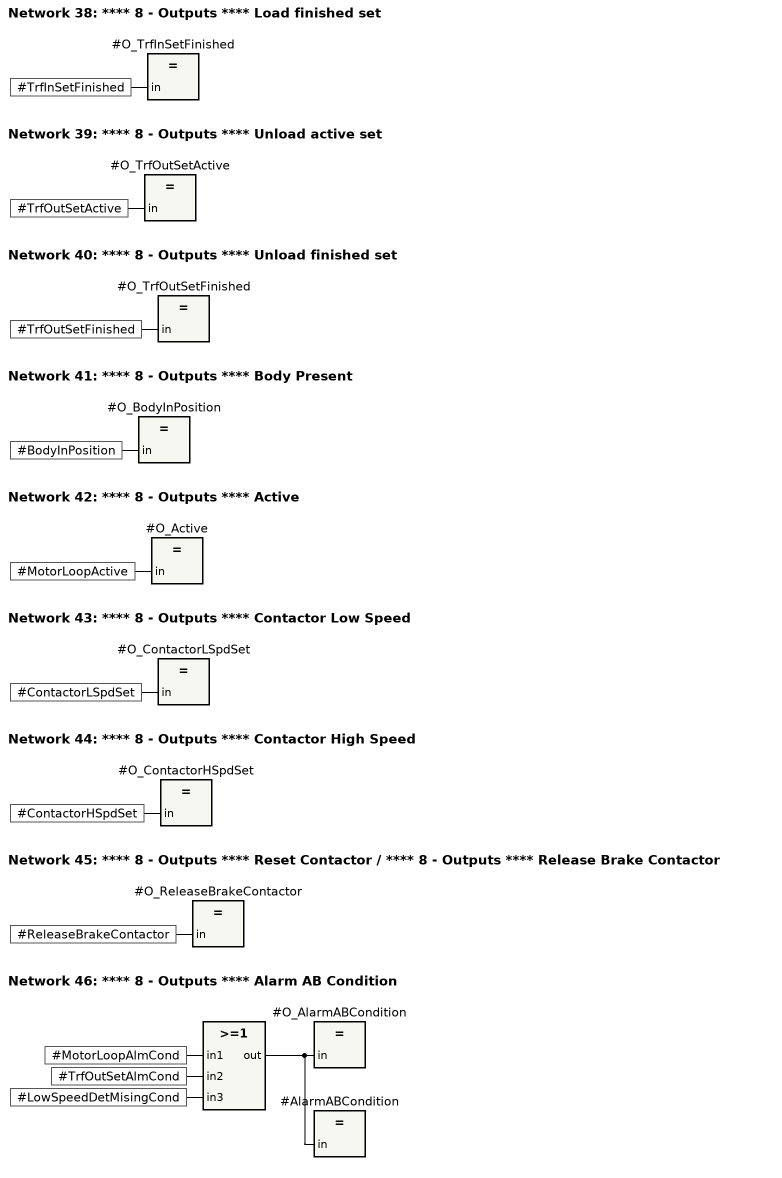
   #O_TrfInSetFinished := #TrfInSetFinished;
END_REGION

REGION Network 39: **** 8 - Outputs **** Unload active set
   // Unload active set
   #O_TrfOutSetActive := #TrfOutSetActive;
END_REGION

REGION Network 40: **** 8 - Outputs **** Unload finished set
   // Unload finished set
   #O_TrfOutSetFinished := #TrfOutSetFinished;
END_REGION

REGION Network 41: **** 8 - Outputs **** Body Present
   // Body present
   #O_BodyInPosition := #BodyInPosition;
END_REGION

REGION Network 42: **** 8 - Outputs **** Active
   // Active
   #O_Active := #MotorLoopActive;
END_REGION

REGION Network 43: **** 8 - Outputs **** Contactor Low Speed
   // Contactor Low Speed
   #O_ContactorLSpdSet := #ContactorLSpdSet;
END_REGION

REGION Network 44: **** 8 - Outputs **** Contactor High Speed
   // Contactor High Speed
   #O_ContactorHSpdSet := #ContactorHSpdSet;
END_REGION

REGION Network 45: **** 8 - Outputs **** Reset Contactor / **** 8 - Outputs **** Release Brake Contactor
   // Reset Contactor / Release Brake Contactor
   #O_ReleaseBrakeContactor := #ReleaseBrakeContactor;
END_REGION

REGION Network 46: **** 8 - Outputs **** Alarm AB Condition
   // Alarm AB Condition
   #O_AlarmABCondition := #MotorLoopAlmCond OR #TrfOutSetAlmCond OR #LowSpeedDetMisingCond;
   #AlarmABCondition := #O_AlarmABCondition;
END_REGION

REGION Network 47: **** 8 - Outputs **** Led
   // Led
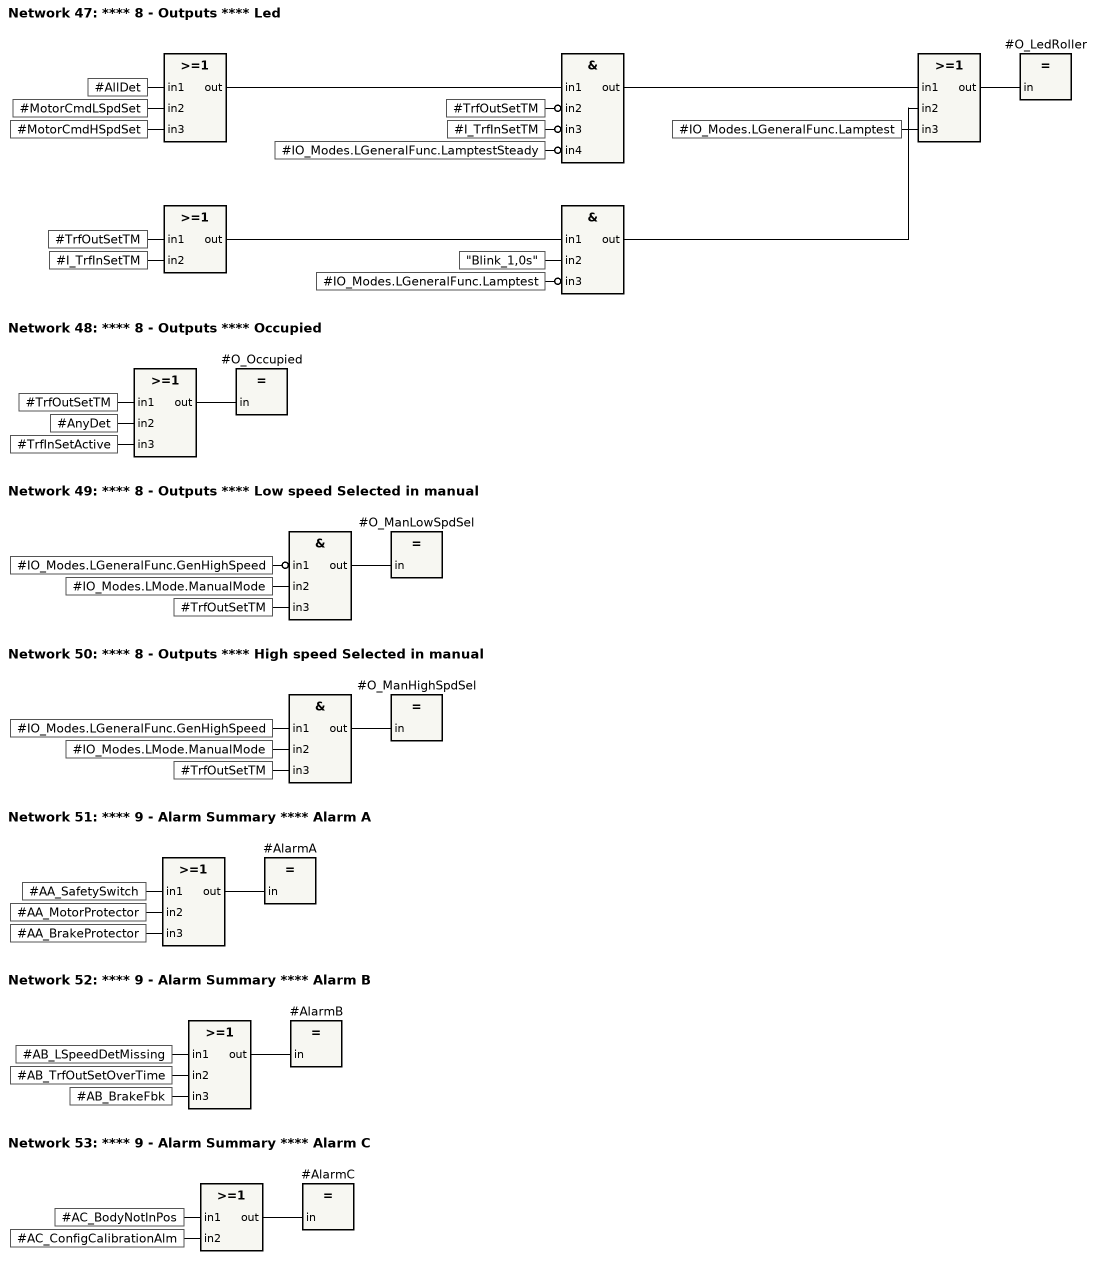
   #O_LedRoller := ((#AllDet OR #MotorCmdLSpdSet OR #MotorCmdHSpdSet) AND NOT #TrfOutSetTM AND NOT #I_TrfInSetTM AND NOT #IO_Modes.LGeneralFunc.LamptestSteady) OR ((#TrfOutSetTM OR #I_TrfInSetTM) AND "Blink_1,0s" AND NOT #IO_Modes.LGeneralFunc.Lamptest) OR #IO_Modes.LGeneralFunc.Lamptest;
END_REGION

REGION Network 48: **** 8 - Outputs **** Occupied
   // Occupied
   #O_Occupied := #TrfOutSetTM OR #AnyDet OR #TrfInSetActive;
END_REGION

REGION Network 49: **** 8 - Outputs **** Low speed Selected in manual
   #O_ManLowSpdSel := NOT #IO_Modes.LGeneralFunc.GenHighSpeed AND #IO_Modes.LMode.ManualMode AND #TrfOutSetTM;
END_REGION

REGION Network 50: **** 8 - Outputs **** High speed Selected in manual
   #O_ManHighSpdSel := #IO_Modes.LGeneralFunc.GenHighSpeed AND #IO_Modes.LMode.ManualMode AND #TrfOutSetTM;
END_REGION

REGION Network 51: **** 9 - Alarm Summary **** Alarm A
   // Alarm A
   #AlarmA := #AA_SafetySwitch OR #AA_MotorProtector OR #AA_BrakeProtector;
END_REGION

REGION Network 52: **** 9 - Alarm Summary **** Alarm B
   // Alarm B
   #AlarmB := #AB_LSpeedDetMissing OR #AB_TrfOutSetOverTime OR #AB_BrakeFbk;
END_REGION

REGION Network 53: **** 9 - Alarm Summary **** Alarm C
   // Alarm C
   #AlarmC := #AC_BodyNotInPos OR #AC_ConfigCalibrationAlm;
END_REGION

REGION Network 54: **** 9 - Alarm Summary **** Alarm D
   // Alarm D
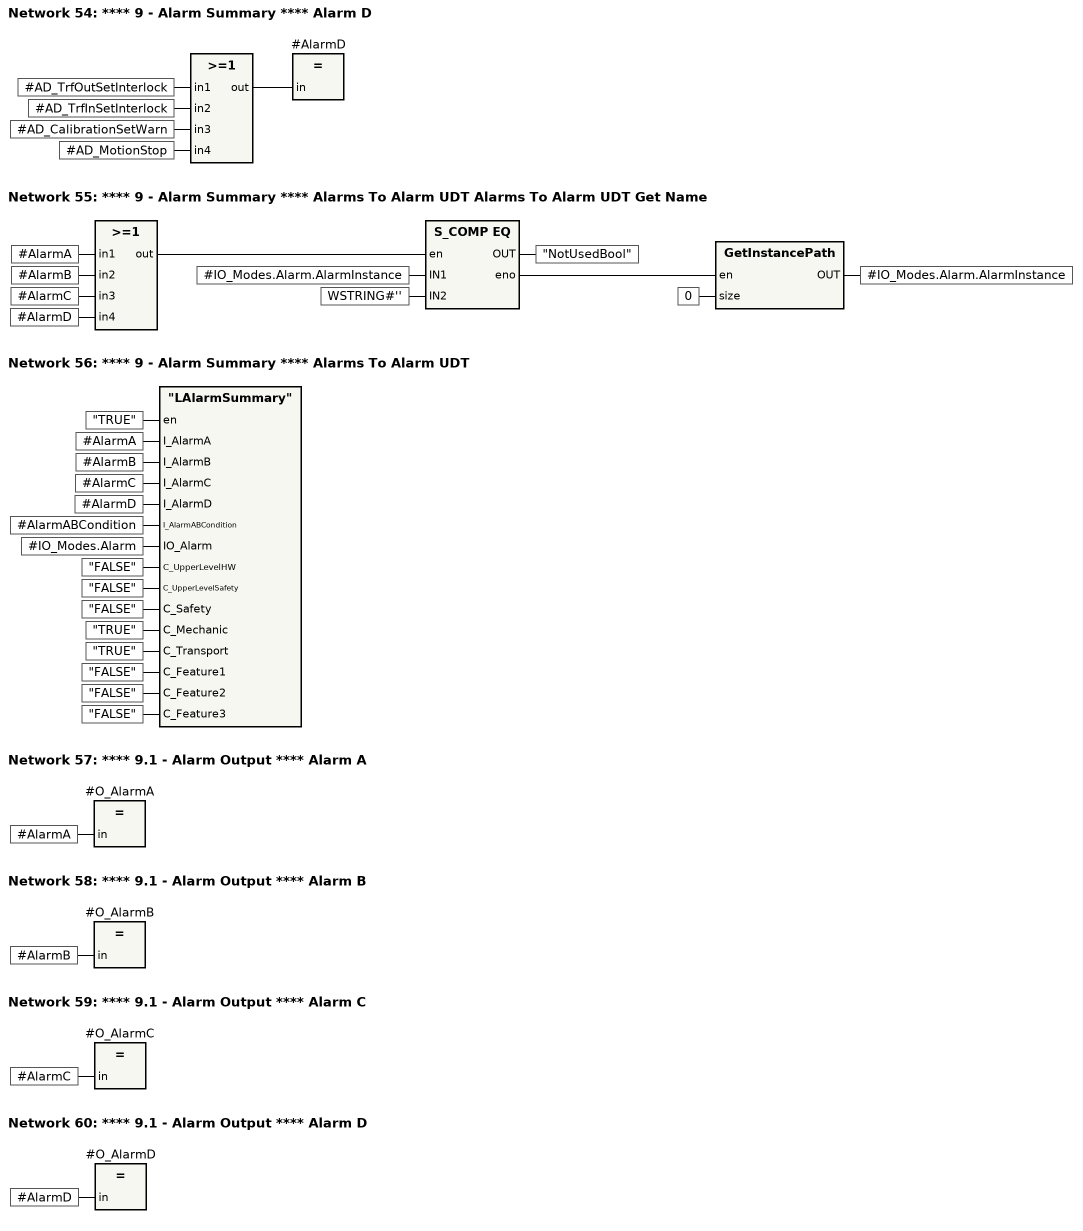
   #AlarmD := #AD_TrfOutSetInterlock OR #AD_TrfInSetInterlock OR #AD_CalibrationSetWarn OR #AD_MotionStop;
END_REGION

REGION Network 55: **** 9 - Alarm Summary **** Alarms To Alarm UDT Alarms To Alarm UDT Get Name
   // Alarm / Alarm D
   S_COMP(EN := #AlarmA OR #AlarmB OR #AlarmC OR #AlarmD,
          IN1 := #IO_Modes.Alarm.AlarmInstance,
          IN2 := WSTRING#'',
          OUT => "NotUsedBool",
          ENO => #_w1);
   IF #_w1 THEN GetInstancePath(size := 0, OUT => #IO_Modes.Alarm.AlarmInstance); END_IF;
END_REGION

REGION Network 56: **** 9 - Alarm Summary **** Alarms To Alarm UDT
   // Alarm / Alarm D
   IF "TRUE" THEN
       "LAlarmSummary"(I_AlarmA := #AlarmA,
                       I_AlarmB := #AlarmB,
                       I_AlarmC := #AlarmC,
                       I_AlarmD := #AlarmD,
                       I_AlarmABCondition := #AlarmABCondition,
                       IO_Alarm := #IO_Modes.Alarm,
                       C_UpperLevelHW := "FALSE",
                       C_UpperLevelSafety := "FALSE",
                       C_Safety := "FALSE",
                       C_Mechanic := "TRUE",
                       C_Transport := "TRUE",
                       C_Feature1 := "FALSE",
                       C_Feature2 := "FALSE",
                       C_Feature3 := "FALSE");
   END_IF;
END_REGION

REGION Network 57: **** 9.1 - Alarm Output **** Alarm A
   // Alarm A
   #O_AlarmA := #AlarmA;
END_REGION

REGION Network 58: **** 9.1 - Alarm Output **** Alarm B
   // Alarm B
   #O_AlarmB := #AlarmB;
END_REGION

REGION Network 59: **** 9.1 - Alarm Output **** Alarm C
   // Alarm C
   #O_AlarmC := #AlarmC;
END_REGION

REGION Network 60: **** 9.1 - Alarm Output **** Alarm D
   // Alarm D
   #O_AlarmD := #AlarmD;
END_REGION

REGION Network 61: **** 9.2 - Alarm DWord**** Alarm To DWord
   // Alarm To Word
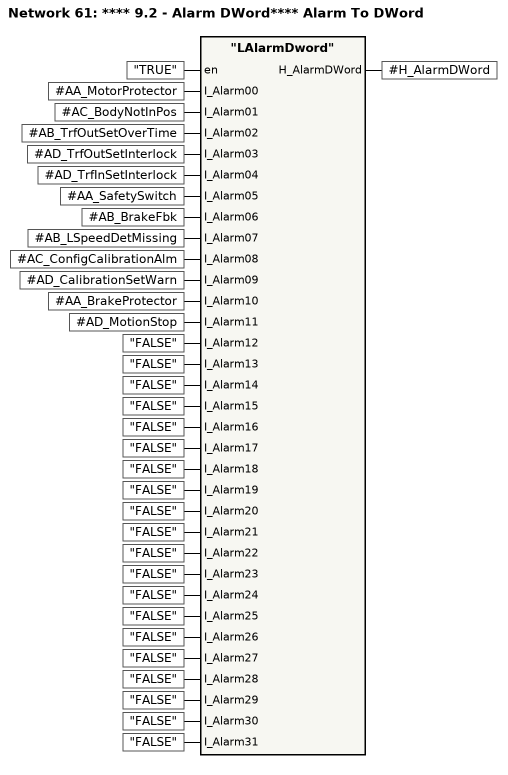
   IF "TRUE" THEN
       "LAlarmDword"(I_Alarm00 := #AA_MotorProtector,
                     I_Alarm01 := #AC_BodyNotInPos,
                     I_Alarm02 := #AB_TrfOutSetOverTime,
                     I_Alarm03 := #AD_TrfOutSetInterlock,
                     I_Alarm04 := #AD_TrfInSetInterlock,
                     I_Alarm05 := #AA_SafetySwitch,
                     I_Alarm06 := #AB_BrakeFbk,
                     I_Alarm07 := #AB_LSpeedDetMissing,
                     I_Alarm08 := #AC_ConfigCalibrationAlm,
                     I_Alarm09 := #AD_CalibrationSetWarn,
                     I_Alarm10 := #AA_BrakeProtector,
                     I_Alarm11 := #AD_MotionStop,
                     I_Alarm12 := "FALSE",
                     I_Alarm13 := "FALSE",
                     I_Alarm14 := "FALSE",
                     I_Alarm15 := "FALSE",
                     I_Alarm16 := "FALSE",
                     I_Alarm17 := "FALSE",
                     I_Alarm18 := "FALSE",
                     I_Alarm19 := "FALSE",
                     I_Alarm20 := "FALSE",
                     I_Alarm21 := "FALSE",
                     I_Alarm22 := "FALSE",
                     I_Alarm23 := "FALSE",
                     I_Alarm24 := "FALSE",
                     I_Alarm25 := "FALSE",
                     I_Alarm26 := "FALSE",
                     I_Alarm27 := "FALSE",
                     I_Alarm28 := "FALSE",
                     I_Alarm29 := "FALSE",
                     I_Alarm30 := "FALSE",
                     I_Alarm31 := "FALSE",
                     H_AlarmDWord => #H_AlarmDWord);
   END_IF;
END_REGION
END_FUNCTION_BLOCK
